(* CODESYS project sensata_pressuretransducers.library
   Company: Sensata Technologies
   Version: 0.0.1
   DocFormat: reStructuredText
   Placeholder: Sensata_PressureTransducers
   Title: Sensata_PressureTransducers

Project tree, tasks and I/O mapping:
  libraries: Sensata_Common, * (Sensata Technologies); Sensata_Utilities, * (Sensata Technologies); Tc2_Standard, * (Beckhoff Automation GmbH); Tc2_System, * (Beckhoff Automation GmbH); Tc2_Utilities, * (Beckhoff Automation GmbH); Tc3_Module, * (Beckhoff Automation GmbH)
  Abstract/
    function block FB_PressureTransducer [ST]: M_GetAlicatFlowData, M_GetPressure
  Concrete/
    Agilent/
      AgilentVacuumGauge/
        function block FB_AgilentVacuumGauge [ST]: M_Connect, M_Disconnect, M_GetConnectStatus, P_bConnectBusy, P_bConnected, P_strDescription, P_strMake, P_strModel, P_strVersion, M_GetPressure, A_CommandRecovery, M_RouterHelper
      data type E_Agilent_Error
    Alicat/
      AlicatAbsolute/
        function block FB_AlicatAbsolute [ST]: M_GetAlicatAbsData, M_LockDisplay, M_UnlockDisplay, M_Connect, M_Disconnect, M_GetConnectStatus, P_bConnectBusy, P_bConnected, P_strDescription, P_strMake, P_strModel, P_strVersion, M_GetPressure, A_CommandRecovery, M_RouterHelper
      AlicatDifferential/
        function block FB_AlicatDifferential [ST]: M_GetAlicatDiffData, M_LockDisplay, M_Tare, M_UnlockDisplay, M_Connect, M_Disconnect, M_GetConnectStatus, P_bConnectBusy, P_bConnected, P_strDescription, P_strMake, P_strModel, P_strVersion, M_GetPressure, A_CommandRecovery, M_RouterHelper
      AlicatFlowMeter/
        function block FB_AlicatFlowMeter [ST]: M_GetAlicatFlowData, M_LockDisplay, M_Tare, M_UnlockDisplay, M_Connect, M_Disconnect, M_GetConnectStatus, P_bConnectBusy, P_bConnected, P_strDescription, P_strMake, P_strModel, P_strVersion, M_GetPressure, A_CommandRecovery, M_RouterHelper
      data type E_Alicat_Error
    Structures/
      data type ST_AlicatAbsoluteDataFrame
      data type ST_AlicatDifferentialDataFrame
      data type ST_AlicatFlowMeter
      data type ST_SerialDataFrame
  Interfaces/
    interface I_PressureSensing: M_GetPressure
  Project Information/
    function F_GetCompany [ST]
    function F_GetTitle [ST]
    function F_GetVersion [ST]
  Version/
    global variables Global_Version
*)

// Concrete/Agilent/E_Agilent_Error
{attribute 'qualified_only'}
{attribute 'strict'}
TYPE E_Agilent_Error :
(
	None := 0,
	
	CommandRouterError			:= 0100,  // Error on the command router FB
	CommandFault 				:= 0101, // Command failed to execute
	
	FailedToConnect 			:= 0200, // Connect command failed
	FailedToDisconnect 			:= 0201, // Disonnect command failed
	FailedToGetConnectStatus 	:= 0202, // GetConnectStatus command failed
	
	FailedToReadSerialData		:= 0203,   // ReadSerialDataFrame from Agilent failed
	
	FailedToLoadProgram			:= 0300, // LoadProgram command failed
	FailedToGetCurrentProgram	:= 0301, // GetCurrentProgram command failed
	FailedToStartProgram		:= 0302, // StartProgram command failed
	FailedToStopProgram			:= 0303, // StopProgram command failed
	FailedToPauseProgram		:= 0304, // PauseProgram command failed
	FailedToGetProgramState		:= 0305, // GetProgramState command failed
	
	FailedToEnable				:= 0400, // Enable command failed
	FailedToDisable				:= 0401, // Disable command failed
	FailedToGetEnableStatus		:= 0402, // GetEnableStatus command failed
	
	FailedToPowerOn				:= 0500, // PowerOn command failed
	FailedToPowerOff			:= 0501, // PowerOff command failed
	FailedToGetPowerStatus		:= 0502, // GetPowerStatus command failed
	
	FailedToReset				:= 0600, // Reset command failed

	FailedToGetSafetyStatus		:= 0700 // GetSafetyStatus command failed
) UDINT;
END_TYPE

// Concrete/Alicat/E_Alicat_Error
{attribute 'qualified_only'}
{attribute 'strict'}
TYPE E_Alicat_Error :
(
	None := 0,
	
	CommandRouterError			:= 0100,  // Error on the command router FB
	CommandFault 				:= 0101, // Command failed to execute
	
	FailedToConnect 			:= 0200, // Connect command failed
	FailedToDisconnect 			:= 0201, // Disonnect command failed
	FailedToGetConnectStatus 	:= 0202, // GetConnectStatus command failed
	
	FailedToReadSerialData		:= 0203,   // ReadSerialDataFrame from Alicat failed
	FailedToLockDisplay			:= 0204,   // LockDisplay of AlicatDevice failed
	FailedToUnlockDisplay		:= 0205,   // UnlockDisplay of AlicatDevice failed
	FailedToTareDifferentialGauge := 0206, //Taring Differential Pressure Transducer failed
	FailedToTareFlowMeter 		:= 0207,   //Taring Flow Meter failed
	
	FailedToLoadProgram			:= 0300, // LoadProgram command failed
	FailedToGetCurrentProgram	:= 0301, // GetCurrentProgram command failed
	FailedToStartProgram		:= 0302, // StartProgram command failed
	FailedToStopProgram			:= 0303, // StopProgram command failed
	FailedToPauseProgram		:= 0304, // PauseProgram command failed
	FailedToGetProgramState		:= 0305, // GetProgramState command failed
	
	FailedToEnable				:= 0400, // Enable command failed
	FailedToDisable				:= 0401, // Disable command failed
	FailedToGetEnableStatus		:= 0402, // GetEnableStatus command failed
	
	FailedToPowerOn				:= 0500, // PowerOn command failed
	FailedToPowerOff			:= 0501, // PowerOff command failed
	FailedToGetPowerStatus		:= 0502, // GetPowerStatus command failed
	
	FailedToReset				:= 0600, // Reset command failed

	FailedToGetSafetyStatus		:= 0700 // GetSafetyStatus command failed
) UDINT;
END_TYPE

// Concrete/Structures/ST_AlicatAbsoluteDataFrame
TYPE ST_AlicatAbsoluteDataFrame :
STRUCT
	strDeviceID : STRING;
	lrAbsPressure : LREAL;
	strStatusCode : STRING;	
END_STRUCT
END_TYPE

// Concrete/Structures/ST_AlicatDifferentialDataFrame
TYPE ST_AlicatDifferentialDataFrame :
STRUCT
	strDeviceID : STRING;
	lrDiffPressure : LREAL;
	strStatusCode : STRING;	
END_STRUCT
END_TYPE

// Concrete/Structures/ST_AlicatFlowMeter
TYPE ST_AlicatFlowMeter :
STRUCT
	strDeviceID     : STRING;
	lrAbsPressure   : LREAL;
	lrTemperature   : LREAL;
	lrVolFlowRate   : LREAL;
	lrMassFlowRate  : LREAL;
	lrTotalizedFlow : LREAL;
	strGasSelect    : STRING;
	strStatusCode   : STRING;
END_STRUCT
END_TYPE

// Concrete/Structures/ST_SerialDataFrame
TYPE ST_SerialDataFrame :
STRUCT
	stAlicatAbs : ST_AlicatAbsoluteDataFrame;
	stAlicatDiff : ST_AlicatDifferentialDataFrame;
	stAlicatFlow : ST_AlicatFlowMeter;
END_STRUCT
END_TYPE

// Version/Global_Version
{attribute 'TcGenerated'}
{attribute 'no-analysis'}
{attribute 'linkalways'}
// This function has been automatically generated from the project information.
VAR_GLOBAL CONSTANT
	{attribute 'const_non_replaced'}
	stLibVersion_Sensata_PressureTransducers : ST_LibVersion := (iMajor := 0, iMinor := 0, iBuild := 1, iRevision := 0, nFlags := 0, sVersion := '0.0.1');
END_VAR

// Abstract/FB_PressureTransducer
FUNCTION_BLOCK FB_PressureTransducer EXTENDS FB_Device IMPLEMENTS I_PressureSensing
VAR_INPUT
END_VAR
VAR_OUTPUT
END_VAR
VAR
END_VAR

METHOD M_GetAlicatFlowData : BOOL

VAR_OUTPUT
		(*_output/input_datatypeName*)
	_out_lrealPressure	   : LREAL;
	_out_lrealTotFlow      : LREAL;
	_out_lrealMassFlowRate : LREAL;
	_out_lrealVolFlowRate  : LREAL;
	_out_stResult : ST_SerialDataFrame;
END_VAR
M_GetAlicatFlowData := TRUE;
THIS^.M_LogWarning('M_GetAlicatFlowData not implemented');
END_METHOD

METHOD M_GetPressure : BOOL
VAR_OUTPUT
	(*_output/input_datatypeName*)
	_out_lrealPressure	: LREAL;
END_VAR
M_GetPressure := TRUE;
THIS^.M_LogWarning('M_GetPressure not implemented');
END_METHOD

END_FUNCTION_BLOCK

// Interfaces/I_PressureSensing
INTERFACE I_PressureSensing

METHOD M_GetPressure : BOOL
VAR_INPUT
END_VAR
VAR_OUTPUT
	_out_lrealPressure : LREAL; //_output/input_datatypeName
END_VAR
END_METHOD

END_INTERFACE

// Concrete/Agilent/AgilentVacuumGauge/FB_AgilentVacuumGauge
FUNCTION_BLOCK FB_AgilentVacuumGauge EXTENDS FB_PressureTransducer IMPLEMENTS I_PressureSensing, I_Connectable, I_DeviceInfo
VAR_INPUT
	in_fbApi : REFERENCE TO FB_CommandRouter;
END_VAR
VAR_OUTPUT
END_VAR
VAR
	//Copied all the variables from UReSeries program - still not sure which all we need
	bConnected: BOOL; // Value of P_bConnected
	bEnabled: BOOL; // Value of P_bEnabled
	bPoweredOn: BOOL; // Value of P_bPoweredOn
	strLoadedProgram: STRING(255); // Value of P_strLoadedProgram
	enumProgramState: E_PROGRAMSTATE; // Value of P_enumProgramState
	bRouterBusy: BOOL; // TRUE while M_RouterHelper is being used by a method
	bResetBusy: BOOL; // Value of P_bResetBusy
	
	//ST Adding parameters below
	bDisconnected: BOOL;
	bGetPressureSuccessful: BOOL;
	
	//Command Steps
	intGetPressureStep		 : INT;
	intConnectStep	  		 : INT;
	intDisconnectStep 		 : INT;
	intRouterHelperStep		: INT;
		
	//CommandBusy Bits
	bGetPressureBusy 	   : BOOL;
	bConnectBusy	 	   : BOOL;
	bDisconnectBusy  	   : BOOL;
	bRouterHelperBusy	   : BOOL;
END_VAR

A_CommandRecovery();

(* This method should establish any external connections required to use the
	functions of the device, and return TRUE and set P_bConnected to TRUE once
	connected. *)
METHOD M_Connect : BOOL
VAR CONSTANT
	_strCOMMAND_NAME : T_MaxString	:= 'Connect'; // Name of the API method
	_timeCOMMAND_TIMEOUT : TIME		:= T#100S; // Max time to receive API response
	_strSTART_MSG : T_MaxString		:= 'Connecting'; // Prints when method starts
	_strEND_MSG : T_MaxString		:= 'Connected'; // Prints when method finishes
	_udintERROR_ID : UDINT			:= E_Agilent_Error.FailedToConnect; // Error ID to set if command fails
	_strERROR_MSG : T_MaxString		:= 'Failed to connect to Agilent Vacuum Gauge!'; // Error message to set if command fails
END_VAR
VAR_INST
	_inst_arrParams: T_ApiParameterList; // Parameters array
	_inst_arrOutputs: T_ApiParameterList; // Outputs array
	_inst_strRet: T_ApiParamValue; // Return string from the router
	_inst_intStep: INT; // Current method step
	_inst_fbParams: FB_ApiParamBuilder; // Parameter builder FB
END_VAR
VAR
	_bComplete: BOOL; // True if the routing finishes
	_intRet: INT; // Return string converted to an integer
	_bResult : BOOL; // Output of the method
END_VAR
_inst_intStep := intConnectStep;
bConnectBusy  := TRUE;

_bResult := FALSE;
CASE _inst_intStep OF
	0: // Wait for no error and router not busy
		IF NOT THIS^.P_bError AND NOT bRouterBusy THEN
			bRouterBusy := TRUE;
			_inst_intStep := _inst_intStep + 10;
		END_IF
		
	10: // Initialize parameters
		THIS^.M_LogMessage(_strSTART_MSG);
		_inst_fbParams.M_ClearParameters();
		// ADD ANY PARAMETERS HERE
		_inst_fbParams.M_OutputToParameterList(_inst_arrParams);
		_inst_intStep := _inst_intStep + 10;
		
	20: // Route the command
		_bComplete := M_RouterHelper(
			_in_strMethodName := _strCOMMAND_NAME, 
			_in_timeTimeout := _timeCOMMAND_TIMEOUT,
			_inout_arrParams := _inst_arrParams,
			_inout_arrOutputs := _inst_arrOutputs,
			_out_strReturnValue=>_inst_strRet);
		
		// If route completed, move to next step
		IF _bComplete THEN
			_inst_intStep := _inst_intStep + 10;
			bRouterBusy := FALSE;
		ELSIF THIS^.P_bError THEN
			_inst_intStep := 0;
			bRouterBusy := FALSE;
		END_IF
		
	30: // Parse results
		_intRet := STRING_TO_INT(_inst_strRet);
		IF _intRet > 0 THEN
			_bResult := TRUE;
			THIS^.M_LogMessage(_strEND_MSG);
			// DO ANY PARSING HERE
			bConnected := TRUE;
			
		// Set error if command failed
		ELSE
			THIS^.M_SetError(_udintERROR_ID, _strERROR_MSG);
		END_IF
		
		// Go back to start
		_inst_intStep := 0;
END_CASE
M_Connect := _bResult;
intConnectStep := _inst_intStep;
END_METHOD

(* This method should break any connections established by M_Connect. It should
	immediately set P_bConnected to false unless all connections are known to
	be still active, and return TRUE once those connections are all fully
	disconnected. *)
METHOD M_Disconnect : BOOL
VAR CONSTANT
	_strCOMMAND_NAME : T_MaxString	:= 'Disconnect'; // Name of the API method
	_timeCOMMAND_TIMEOUT : TIME		:= T#30S; // Max time to receive API response
	_strSTART_MSG : T_MaxString		:= 'Disconnecting'; // Prints when method starts
	_strEND_MSG : T_MaxString		:= 'Disconnected'; // Prints when method finishes
	_udintERROR_ID : UDINT			:= E_Agilent_Error.FailedToDisconnect; // Error ID to set if command fails
	_strERROR_MSG : T_MaxString		:= 'Failed to disconnect from AgilentVacuumGauge!'; // Error message to set if command fails
END_VAR
VAR_INST
	_inst_arrParams: T_ApiParameterList; // Parameters array
	_inst_arrOutputs: T_ApiParameterList; // Outputs array
	_inst_strRet: T_ApiParamValue; // Return string from the router
	_inst_intStep: INT; // Current method step
	_inst_fbParams: FB_ApiParamBuilder; // Parameter builder FB
END_VAR
VAR
	_bComplete: BOOL; // True if the routing finishes
	_intRet: INT; // Return string converted to an integer
	_bResult : BOOL; // Output of the method
END_VAR
_inst_intStep := intDisconnectStep;
bDisconnectBusy := TRUE;

_bResult := FALSE;
CASE _inst_intStep OF
	0: // Wait for no error and router not busy
		IF NOT THIS^.P_bError AND NOT bRouterBusy THEN
			bRouterBusy := TRUE;
			_inst_intStep := _inst_intStep + 10;
		END_IF
		
	10: // Initialize parameters
		THIS^.M_LogMessage(_strSTART_MSG);
		_inst_fbParams.M_ClearParameters();
		// ADD ANY PARAMETERS HERE
		_inst_fbParams.M_OutputToParameterList(_inst_arrParams);
		_inst_intStep := _inst_intStep + 10;
		
	20: // Route the command
		_bComplete := M_RouterHelper(
			_in_strMethodName := _strCOMMAND_NAME, 
			_in_timeTimeout := _timeCOMMAND_TIMEOUT,
			_inout_arrParams := _inst_arrParams,
			_inout_arrOutputs := _inst_arrOutputs,
			_out_strReturnValue=>_inst_strRet);
		
		// If route completed, move to next step
		IF _bComplete THEN
			_inst_intStep := _inst_intStep + 10;
			bRouterBusy := FALSE;
		ELSIF THIS^.P_bError THEN
			_inst_intStep := 0;
			bRouterBusy := FALSE;
		END_IF
		
	30: // Parse results
		_intRet := STRING_TO_INT(_inst_strRet);
		IF _intRet > 0 THEN
			_bResult := TRUE;
			THIS^.M_LogMessage(_strEND_MSG);
			// DO ANY PARSING HERE
			bConnected := FALSE;
			
		// Set error if command failed
		ELSE
			THIS^.M_SetError(_udintERROR_ID, _strERROR_MSG);
		END_IF
		
		// Go back to start
		_inst_intStep := 0;
END_CASE
M_Disconnect := _bResult;
intDisconnectStep := _inst_intStep;
END_METHOD

(* This method should explicitly check the connection status of the device.
	Once the connection status is known, this method should return TRUE.
	If this method fails, P_bConnected should be set to FALSE since the device
	is not absolutely known to still be connected. *)
METHOD M_GetConnectStatus : BOOL
VAR_OUTPUT
	(* This should return TRUE if all connections required to make the device
		function properly are known to be connected, and FALSE otherwise. *)
	bConnected	: BOOL;
END_VAR
bConnected := P_bConnected;
M_GetConnectStatus := TRUE;
THIS^.M_LogWarning('Get connect status not implemented in FB_AgilentVacuumGauge!');
END_METHOD

(* This property should be TRUE while any method in this interface is actively
	executing, or FALSE otherwise. *)
PROPERTY P_bConnectBusy : BOOL
GET
END_GET
END_PROPERTY

(* This should be set to TRUE if M_Connect is successful or M_GetConnectStatus
	determines the device to be connected, and set to FALSE if M_Disconnect is
	called at all, M_GetConnectStatus fails, or M_GetConnectStatus determines
	the device to be not connected. *)
PROPERTY P_bConnected : BOOL
GET
END_GET
END_PROPERTY

PROPERTY P_strDescription : Sensata_Common.T_MaxString
GET
END_GET
END_PROPERTY

PROPERTY P_strMake : Sensata_Common.T_MaxString
GET
END_GET
END_PROPERTY

PROPERTY P_strModel : Sensata_Common.T_MaxString
GET
END_GET
END_PROPERTY

PROPERTY P_strVersion : Sensata_Common.T_MaxString
GET
END_GET
END_PROPERTY

METHOD M_GetPressure : BOOL
VAR_OUTPUT
	(*_output/input_datatypeName*)
	_out_lrealPressure	: LREAL;
END_VAR
VAR CONSTANT
	_strCOMMAND_NAME : T_MaxString	:= 'GetPressure'; // Name of the API method
	_timeCOMMAND_TIMEOUT : TIME		:= T#5S; // Max time to receive API response
	_strSTART_MSG : T_MaxString		:= 'Reading Pressure Value'; // Prints when method starts
	_strEND_MSG : T_MaxString		:= 'Pressure Read'; // Prints when method finishes
	_udintERROR_ID : UDINT			:= E_Agilent_Error.FailedToReadSerialData; // Error ID to set if command fails
	_strERROR_MSG : T_MaxString		:= 'Failed to read serial data and hence pressure!'; // Error message to set if command fails
END_VAR
VAR_INST
	_inst_arrParams: T_ApiParameterList; // Parameters array
	_inst_arrOutputs: T_ApiParameterList; // Outputs array
	_inst_strRet: T_ApiParamValue; // Return string from the router
	_inst_intStep: INT; // Current method step
	_inst_fbParams: FB_ApiParamBuilder; // Parameter builder FB
END_VAR
VAR
	_bComplete: BOOL; // True if the routing finishes
	_intRet: INT; // Return string converted to an integer
	_bResult : BOOL; // Output of the method
END_VAR
_inst_intStep := intGetPressureStep;
bGetPressureBusy := TRUE;

_bResult := FALSE;
CASE _inst_intStep OF
	0: // Wait for no error and router not busy
		IF NOT THIS^.P_bError AND NOT bRouterBusy THEN
			bRouterBusy := TRUE;
			_inst_intStep := _inst_intStep + 10;
		END_IF
		
	10: // Initialize parameters
		THIS^.M_LogMessage(_strSTART_MSG);
		_inst_fbParams.M_ClearParameters();
		// ADD ANY PARAMETERS HERE
		_inst_fbParams.M_OutputToParameterList(_inst_arrParams);
		_inst_intStep := _inst_intStep + 10;
		
	20: // Route the command
		_bComplete := M_RouterHelper(
			_in_strMethodName := _strCOMMAND_NAME, 
			_in_timeTimeout := _timeCOMMAND_TIMEOUT,
			_inout_arrParams := _inst_arrParams,
			_inout_arrOutputs := _inst_arrOutputs,
			_out_strReturnValue=>_inst_strRet);
		
		// If route completed, move to next step
		IF _bComplete THEN
			_inst_intStep := _inst_intStep + 10;
			bRouterBusy := FALSE;
		ELSIF THIS^.P_bError THEN
			_inst_intStep := 0;
			bRouterBusy := FALSE;
		END_IF
		
	30: // Parse results
		_intRet := STRING_TO_INT(_inst_strRet);
		IF _intRet > 0 THEN
			_bResult := TRUE;
			THIS^.M_LogMessage(_strEND_MSG);
			// DO ANY PARSING HERE
			_out_lrealPressure := _inst_fbParams.M_ParseDouble(_inst_fbParams.M_GetParameter('Pressure'));
//			_inst_fbParams.M_LoadFromParameterList(_inst_arrOutputs);
//			bEnabled := _inst_fbParams.M_ParseBool(_inst_fbParams.M_GetParameter('enabled'));
//			THIS^.bEnabled := bEnabled;			
			
		// Set error if command failed
		ELSE
			THIS^.M_SetError(_udintERROR_ID, _strERROR_MSG);
		END_IF
		
		// Go back to start
		_inst_intStep := 0;
END_CASE
M_GetPressure := _bResult;
intGetPressureStep := _inst_intStep;
END_METHOD

ACTION A_CommandRecovery:
IF NOT bGetPressureBusy AND intGetPressureStep > 0 THEN
	intGetPressureStep := 0;
	bRouterBusy := FALSE;
	THIS^.M_LogWarning('Get Pressure ended prematurely!');
END_IF
bGetPressureBusy := FALSE;

IF NOT bConnectBusy AND intConnectStep > 0 THEN
	intConnectStep := 0;
	bRouterBusy := FALSE;
	THIS^.M_LogWarning('Connect ended prematurely!');
END_IF
bConnectBusy := FALSE;

IF NOT bDisconnectBusy AND intDisconnectStep > 0 THEN
	intDisconnectStep := 0;
	bRouterBusy := FALSE;
	THIS^.M_LogWarning('Disconnect ended prematurely!');
END_IF
bDisconnectBusy := FALSE;

IF NOT bRouterHelperBusy AND intRouterHelperStep > 0 THEN
	intRouterHelperStep := 0;
	THIS^.M_LogWarning('Router helper ended prematurely!');
END_IF
bRouterHelperBusy := FALSE;
END_ACTION

(*
Sends the given method to the API and receives and partially parses the result.
*)
METHOD PRIVATE M_RouterHelper : BOOL
VAR_INPUT
	(* Name of the method to call. *)
	_in_strMethodName : T_MaxString;
	(* Maximum time to wait for method response. *)
	_in_timeTimeout : TIME;
END_VAR
VAR_IN_OUT
	(* The array of parameters to send to the API. *)
	_inout_arrParams : T_ApiParameterList;
	(* The array that gets populated with any method output data. *)
	_inout_arrOutputs : T_ApiParameterList;
END_VAR
VAR_OUTPUT
	(* JSON string of the method return value. *)
	_out_strReturnValue: T_ApiParamValue;
END_VAR
VAR_INST
	(* Current step. *)
	_inst_intStep: INT;
	(* True if the method executed. *)
	_inst_bExec: BOOL;
	(* Return string of the method. *)
	_inst_strRet: T_ApiParamValue;
END_VAR
VAR
	(* True once the command routing finishes. *)
	_bComplete: BOOL;
	(* True once the API connects. *)
	_bApiConnect: BOOL;
END_VAR
_inst_intStep := intRouterHelperStep;
bRouterHelperBusy := TRUE;

CASE _inst_intStep OF
	0: // Start process only if there is no error on this FB
		IF NOT THIS^.P_bError THEN
			_inst_intStep := 10;
		END_IF
		
	10: // Check if command router connected
		IF NOT in_fbApi.P_bConnected THEN
			_inst_intStep := 20; // Go to API connect step
		ELSE
			_inst_intStep := 30; // Go to route command step
		END_IF
		
	20: // Connect the command router
		_bApiConnect := in_fbApi.M_Connect();
		IF _bApiConnect THEN
			_inst_intStep := _inst_intStep + 10; // Go to next step
		ELSIF in_fbApi.P_bError THEN
			THIS^.M_SetError(E_Agilent_Error.CommandRouterError, 'Error on command router function block while connecting!');
			_inst_intStep := 0; // Go back to start
		END_IF
		
	30:	// Route the command
		_bComplete := in_fbApi.M_RouteCommand(
			_in_strModuleId := in_strUniqueId,
			_in_strMethodName := _in_strMethodName,
			_in_timeTimeout := _in_timeTimeout,
			_inout_arrParameters := _inout_arrParams,
			_inout_arrOutputs := _inout_arrOutputs,
			_out_bCommandExecuted => _inst_bExec,
			_out_strReturnValue => _inst_strRet);
		IF _bComplete THEN
			_inst_intStep := _inst_intStep + 10; // Go to next step
		ELSIF in_fbApi.P_bError THEN
			THIS^.M_SetError(E_Agilent_Error.CommandRouterError, 'Error on command router function block while routing command!');
			_inst_intStep := 0; // Go back to start
		END_IF
		
	40: // Check result then go back to start
		IF NOT _inst_bExec THEN
			THIS^.M_SetError(E_Agilent_Error.CommandFault, 'Method in API failed to execute!');
		ELSE
			_out_strReturnValue := _inst_strRet;
			M_RouterHelper := TRUE;
		END_IF
		_inst_intStep := 0; // Go back to start
END_CASE
intRouterHelperStep := _inst_intStep;
END_METHOD

END_FUNCTION_BLOCK

// Concrete/Alicat/AlicatAbsolute/FB_AlicatAbsolute
FUNCTION_BLOCK FB_AlicatAbsolute EXTENDS FB_PressureTransducer IMPLEMENTS I_PressureSensing, I_Connectable, I_DeviceInfo
VAR_INPUT
	in_fbApi : REFERENCE TO FB_CommandRouter;
END_VAR
VAR_OUTPUT
END_VAR
VAR
	//Copied all the variables from UReSeries program - still not sure which all we need
	bConnected: BOOL; // Value of P_bConnected
	bEnabled: BOOL; // Value of P_bEnabled
	bPoweredOn: BOOL; // Value of P_bPoweredOn
	strLoadedProgram: STRING(255); // Value of P_strLoadedProgram
	enumProgramState: E_PROGRAMSTATE; // Value of P_enumProgramState
	bRouterBusy: BOOL; // TRUE while M_RouterHelper is being used by a method
	bResetBusy: BOOL; // Value of P_bResetBusy
	//ST Adding parameters below
	bDisconnected: BOOL;
	bGetPressureSuccessful: BOOL;
	bGetAlicatDataSuccessful: BOOL;
	bLockDisplaySuccessful: BOOL;
	bUnlockDisplaySuccessful: BOOL;
	
	//Command Steps
	intGetPressureStep		 : INT;
	intConnectStep	  		 : INT;
	intDisconnectStep 		 : INT;
	intGetAlicatAbsDataStep : INT;
	intLockDisplayStep		 : INT;
	intUnlockDisplayStep	 : INT;
	intTareStep			  	 : INT;
	intRouterHelperStep	     : INT;
	
	
	//CommandBusy Bits
	bGetPressureBusy 	   : BOOL;
	bConnectBusy	 	   : BOOL;
	bDisconnectBusy  	   : BOOL;
	bGetAlicatAbsDataBusy  : BOOL;
	bLockDisplayBusy	   : BOOL;
	bUnlockDisplayBusy	   : BOOL;
	bTareBusy			   : BOOL;
	bRouterHelperBusy	   : BOOL;
	
END_VAR

A_CommandRecovery();

(* This method returns the Pressure Value from the Alicat Absolute Pressure Gauge.
Once the Pressure value is obtained, this method must return TRUE*)
METHOD M_GetAlicatAbsData : BOOL
VAR_OUTPUT
	(*_output/input_datatypeName*)
	_out_lrealPressure	: LREAL;
	_out_stResult : ST_SerialDataFrame;
END_VAR
VAR CONSTANT
	_strCOMMAND_NAME : T_MaxString	:= 'GetAlicatAbsData'; // Name of the API method
	_timeCOMMAND_TIMEOUT : TIME		:= T#5S; // Max time to receive API response
	_strSTART_MSG : T_MaxString		:= 'Reading Alicat Serial Frame'; // Prints when method starts
	_strEND_MSG : T_MaxString		:= 'Read Alicat Serial Frame successfully'; // Prints when method finishes
	_udintERROR_ID : UDINT			:= E_Alicat_Error.FailedToReadSerialData; // Error ID to set if command fails
	_strERROR_MSG : T_MaxString		:= 'Failed to read Alicat Serial Frame!'; // Error message to set if command fails
END_VAR
VAR_INST
	_inst_arrParams: T_ApiParameterList; // Parameters array
	_inst_arrOutputs: T_ApiParameterList; // Outputs array
	_inst_strRet: T_ApiParamValue; // Return string from the router
	_inst_intStep: INT; // Current method step
	_inst_fbParams: FB_ApiParamBuilder; // Parameter builder FB
END_VAR
VAR
	_bComplete: BOOL; // True if the routing finishes
	_intRet: INT; // Return string converted to an integer
	_bResult : BOOL; // Output of the method
	_pStructPointer : PVOID; // Pointer to the struct
	_pStructPointerAbs : PVOID; 
END_VAR
VAR_INPUT
	
END_VAR
_inst_intStep := intGetAlicatAbsDataStep;
bGetAlicatAbsDataBusy := TRUE;

_bResult := FALSE;
CASE _inst_intStep OF
	0: // Wait for no error and router not busy
		IF NOT THIS^.P_bError AND NOT bRouterBusy THEN
			bRouterBusy := TRUE;
			_inst_intStep := _inst_intStep + 10;
		END_IF
		
	10: // Initialize parameters
		THIS^.M_LogMessage(_strSTART_MSG);
		_inst_fbParams.M_ClearParameters();
		// ADD ANY PARAMETERS HERE
		_inst_fbParams.M_OutputToParameterList(_inst_arrParams);
		_inst_intStep := _inst_intStep + 10;
		
	20: // Route the command
		_bComplete := M_RouterHelper(
			_in_strMethodName := _strCOMMAND_NAME, 
			_in_timeTimeout := _timeCOMMAND_TIMEOUT,
			_inout_arrParams := _inst_arrParams,
			_inout_arrOutputs := _inst_arrOutputs,
			_out_strReturnValue=>_inst_strRet);
		
		// If route completed, move to next step
		IF _bComplete THEN
			_inst_intStep := _inst_intStep + 10;
			bRouterBusy := FALSE;
		ELSIF THIS^.P_bError THEN
			_inst_intStep := 0;
			bRouterBusy := FALSE;
		END_IF
		
	30: // Parse results
		_intRet := STRING_TO_INT(_inst_strRet);
		IF _intRet > 0 THEN
			_bResult := TRUE;
			THIS^.M_LogMessage(_strEND_MSG);
			// DO ANY PARSING HERE
			_pStructPointer := _inst_fbParams.M_GetParameter('alicatAbsDataFrame');	//Because this is the name of the parameter on the API side - type doesn't matter?
			
			_pStructPointerAbs := _inst_fbParams.M_GetStructMember(_pStructPointer, 'AlicatAbsoluteDataFrame');	//Because AlicatAbsoluteDataFrame is a member of the main struct on the API side			
		
			_out_stResult.stAlicatAbs.strDeviceID := _inst_fbParams.M_ParseString(_inst_fbParams.M_GetStructMember(_pStructPointerAbs, 'DeviceID'));
			_out_stResult.stAlicatAbs.lrAbsPressure := _inst_fbParams.M_ParseDouble(_inst_fbParams.M_GetStructMember(_pStructPointerAbs, 'AbsPressure'));
			_out_stResult.stAlicatAbs.strStatusCode := _inst_fbParams.M_ParseString(_inst_fbParams.M_GetStructMember(_pStructPointerAbs, 'StatusCode'));
			
			_out_lrealPressure := _out_stResult.stAlicatAbs.lrAbsPressure;
			
//			_inst_fbParams.M_LoadFromParameterList(_inst_arrOutputs);
//			bConnected := _inst_fbParams.M_ParseBool(_inst_fbParams.M_GetParameter('connected'));
//			THIS^.bConnected := bConnected;
			
		// Set error if command failed
		ELSE
			THIS^.M_SetError(_udintERROR_ID, _strERROR_MSG);
		END_IF
		
		// Go back to start
		_inst_intStep := 0;
END_CASE
M_GetAlicatAbsData := _bResult;
intGetAlicatAbsDataStep := _inst_intStep;
END_METHOD

(* This method returns the status of whether the screen on the device has been locked.
Once the screen is locked, this method must return TRUE*)
METHOD M_LockDisplay : BOOL
VAR_INPUT
END_VAR
VAR CONSTANT
	_strCOMMAND_NAME : T_MaxString	:= 'LockDisplay'; // Name of the API method
	_timeCOMMAND_TIMEOUT : TIME		:= T#2S; // Max time to receive API response
	_strSTART_MSG : T_MaxString		:= 'Locking Alicat Display'; // Prints when method starts
	_strEND_MSG : T_MaxString		:= 'Locked Alicat Display'; // Prints when method finishes
	_udintERROR_ID : UDINT			:= E_Alicat_Error.FailedToLockDisplay; // Error ID to set if command fails
	_strERROR_MSG : T_MaxString		:= 'Failed to lock display!'; // Error message to set if command fails
END_VAR
VAR_INST
	_inst_arrParams: T_ApiParameterList; // Parameters array
	_inst_arrOutputs: T_ApiParameterList; // Outputs array
	_inst_strRet: T_ApiParamValue; // Return string from the router
	_inst_intStep: INT; // Current method step
	_inst_fbParams: FB_ApiParamBuilder; // Parameter builder FB
END_VAR
VAR
	_bComplete: BOOL; // True if the routing finishes
	_intRet: INT; // Return string converted to an integer
	_bResult : BOOL; // Output of the method
END_VAR
_inst_intStep 	 := intLockDisplayStep;
bLockDisplayBusy := TRUE;

_bResult := FALSE;
CASE _inst_intStep OF
	0: // Wait for no error and router not busy
		IF NOT THIS^.P_bError AND NOT bRouterBusy THEN
			bRouterBusy := TRUE;
			_inst_intStep := _inst_intStep + 10;
		END_IF
		
	10: // Initialize parameters
		THIS^.M_LogMessage(_strSTART_MSG);
		_inst_fbParams.M_ClearParameters();
		// ADD ANY PARAMETERS HERE
		_inst_fbParams.M_OutputToParameterList(_inst_arrParams);
		_inst_intStep := _inst_intStep + 10;
		
	20: // Route the command
		_bComplete := M_RouterHelper(
			_in_strMethodName := _strCOMMAND_NAME, 
			_in_timeTimeout := _timeCOMMAND_TIMEOUT,
			_inout_arrParams := _inst_arrParams,
			_inout_arrOutputs := _inst_arrOutputs,
			_out_strReturnValue=>_inst_strRet);
		
		// If route completed, move to next step
		IF _bComplete THEN
			_inst_intStep := _inst_intStep + 10;
			bRouterBusy := FALSE;
		ELSIF THIS^.P_bError THEN
			_inst_intStep := 0;
			bRouterBusy := FALSE;
		END_IF
		
	30: // Parse results
		_intRet := STRING_TO_INT(_inst_strRet);
		IF _intRet > 0 THEN
			_bResult := TRUE;
			THIS^.M_LogMessage(_strEND_MSG);
			// DO ANY PARSING HERE
//			_inst_fbParams.M_LoadFromParameterList(_inst_arrOutputs);
//			bConnected := _inst_fbParams.M_ParseBool(_inst_fbParams.M_GetParameter('connected'));
//			THIS^.bConnected := bConnected;
			
		// Set error if command failed
		ELSE
			THIS^.M_SetError(_udintERROR_ID, _strERROR_MSG);
		END_IF
		
		// Go back to start
		_inst_intStep := 0;
END_CASE
M_LockDisplay := _bResult;
intLockDisplayStep := _inst_intStep;
END_METHOD

(* This method returns the status of whether the screen on the device has been locked.
Once the screen is locked, this method must return TRUE*)
METHOD M_UnlockDisplay : BOOL
VAR_INPUT
END_VAR
VAR CONSTANT
	_strCOMMAND_NAME : T_MaxString	:= 'UnlockDisplay'; // Name of the API method
	_timeCOMMAND_TIMEOUT : TIME		:= T#2S; // Max time to receive API response
	_strSTART_MSG : T_MaxString		:= 'Unlocking Alicat Display'; // Prints when method starts
	_strEND_MSG : T_MaxString		:= 'Unlocked Alicat Display'; // Prints when method finishes
	_udintERROR_ID : UDINT			:= E_Alicat_Error.FailedToUnlockDisplay; // Error ID to set if command fails
	_strERROR_MSG : T_MaxString		:= 'Failed to unlock display!'; // Error message to set if command fails
END_VAR
VAR_INST
	_inst_arrParams: T_ApiParameterList; // Parameters array
	_inst_arrOutputs: T_ApiParameterList; // Outputs array
	_inst_strRet: T_ApiParamValue; // Return string from the router
	_inst_intStep: INT; // Current method step
	_inst_fbParams: FB_ApiParamBuilder; // Parameter builder FB
END_VAR
VAR
	_bComplete: BOOL; // True if the routing finishes
	_intRet: INT; // Return string converted to an integer
	_bResult : BOOL; // Output of the method
END_VAR
_inst_intStep := intUnlockDisplayStep;
bUnlockDisplayBusy := TRUE;

_bResult := FALSE;
CASE _inst_intStep OF
	0: // Wait for no error and router not busy
		IF NOT THIS^.P_bError AND NOT bRouterBusy THEN
			bRouterBusy := TRUE;
			_inst_intStep := _inst_intStep + 10;
		END_IF
		
	10: // Initialize parameters
		THIS^.M_LogMessage(_strSTART_MSG);
		_inst_fbParams.M_ClearParameters();
		// ADD ANY PARAMETERS HERE
		_inst_fbParams.M_OutputToParameterList(_inst_arrParams);
		_inst_intStep := _inst_intStep + 10;
		
	20: // Route the command
		_bComplete := M_RouterHelper(
			_in_strMethodName := _strCOMMAND_NAME, 
			_in_timeTimeout := _timeCOMMAND_TIMEOUT,
			_inout_arrParams := _inst_arrParams,
			_inout_arrOutputs := _inst_arrOutputs,
			_out_strReturnValue=>_inst_strRet);
		
		// If route completed, move to next step
		IF _bComplete THEN
			_inst_intStep := _inst_intStep + 10;
			bRouterBusy := FALSE;
		ELSIF THIS^.P_bError THEN
			_inst_intStep := 0;
			bRouterBusy := FALSE;
		END_IF
		
	30: // Parse results
		_intRet := STRING_TO_INT(_inst_strRet);
		IF _intRet > 0 THEN
			_bResult := TRUE;
			THIS^.M_LogMessage(_strEND_MSG);
			// DO ANY PARSING HERE
//			_inst_fbParams.M_LoadFromParameterList(_inst_arrOutputs);
//			bConnected := _inst_fbParams.M_ParseBool(_inst_fbParams.M_GetParameter('connected'));
//			THIS^.bConnected := bConnected;
			
		// Set error if command failed
		ELSE
			THIS^.M_SetError(_udintERROR_ID, _strERROR_MSG);
		END_IF
		
		// Go back to start
		_inst_intStep := 0;
END_CASE
M_UnlockDisplay := _bResult;
intUnlockDisplayStep := _inst_intStep;
END_METHOD

(* This method should establish any external connections required to use the
	functions of the device, and return TRUE and set P_bConnected to TRUE once
	connected. *)
METHOD M_Connect : BOOL
VAR CONSTANT
	_strCOMMAND_NAME : T_MaxString	:= 'Connect'; // Name of the API method
	_timeCOMMAND_TIMEOUT : TIME		:= T#100S; // Max time to receive API response
	_strSTART_MSG : T_MaxString		:= 'Connecting'; // Prints when method starts
	_strEND_MSG : T_MaxString		:= 'Connected'; // Prints when method finishes
	_udintERROR_ID : UDINT			:= E_Alicat_Error.FailedToConnect; // Error ID to set if command fails
	_strERROR_MSG : T_MaxString		:= 'Failed to connect to Absolute Pressure Transducer!'; // Error message to set if command fails
END_VAR
VAR_INST
	_inst_arrParams: T_ApiParameterList; // Parameters array
	_inst_arrOutputs: T_ApiParameterList; // Outputs array
	_inst_strRet: T_ApiParamValue; // Return string from the router
	_inst_intStep: INT; // Current method step
	_inst_fbParams: FB_ApiParamBuilder; // Parameter builder FB
END_VAR
VAR
	_bComplete: BOOL; // True if the routing finishes
	_intRet: INT; // Return string converted to an integer
	_bResult : BOOL; // Output of the method
END_VAR
_inst_intStep := intConnectStep;
bConnectBusy  := TRUE;

_bResult := FALSE;
CASE _inst_intStep OF
	0: // Wait for no error and router not busy
		IF NOT THIS^.P_bError AND NOT bRouterBusy THEN
			bRouterBusy := TRUE;
			_inst_intStep := _inst_intStep + 10;
		END_IF
		
	10: // Initialize parameters
		THIS^.M_LogMessage(_strSTART_MSG);
		_inst_fbParams.M_ClearParameters();
		// ADD ANY PARAMETERS HERE
		_inst_fbParams.M_OutputToParameterList(_inst_arrParams);
		_inst_intStep := _inst_intStep + 10;
		
	20: // Route the command
		_bComplete := M_RouterHelper(
			_in_strMethodName := _strCOMMAND_NAME, 
			_in_timeTimeout := _timeCOMMAND_TIMEOUT,
			_inout_arrParams := _inst_arrParams,
			_inout_arrOutputs := _inst_arrOutputs,
			_out_strReturnValue=>_inst_strRet);
		
		// If route completed, move to next step
		IF _bComplete THEN
			_inst_intStep := _inst_intStep + 10;
			bRouterBusy := FALSE;
		ELSIF THIS^.P_bError THEN
			_inst_intStep := 0;
			bRouterBusy := FALSE;
		END_IF
		
	30: // Parse results
		_intRet := STRING_TO_INT(_inst_strRet);
		IF _intRet > 0 THEN
			_bResult := TRUE;
			THIS^.M_LogMessage(_strEND_MSG);
			// DO ANY PARSING HERE
			bConnected := TRUE;
			
		// Set error if command failed
		ELSE
			THIS^.M_SetError(_udintERROR_ID, _strERROR_MSG);
		END_IF
		
		// Go back to start
		_inst_intStep := 0;
END_CASE
M_Connect := _bResult;
intConnectStep := _inst_intStep;
END_METHOD

(* This method should break any connections established by M_Connect. It should
	immediately set P_bConnected to false unless all connections are known to
	be still active, and return TRUE once those connections are all fully
	disconnected. *)
METHOD M_Disconnect : BOOL
VAR CONSTANT
	_strCOMMAND_NAME : T_MaxString	:= 'Disconnect'; // Name of the API method
	_timeCOMMAND_TIMEOUT : TIME		:= T#30S; // Max time to receive API response
	_strSTART_MSG : T_MaxString		:= 'Disconnecting'; // Prints when method starts
	_strEND_MSG : T_MaxString		:= 'Disconnected'; // Prints when method finishes
	_udintERROR_ID : UDINT			:= E_Alicat_Error.FailedToDisconnect; // Error ID to set if command fails
	_strERROR_MSG : T_MaxString		:= 'Failed to disconnect from Absolute Pressure Transducer!'; // Error message to set if command fails
END_VAR
VAR_INST
	_inst_arrParams: T_ApiParameterList; // Parameters array
	_inst_arrOutputs: T_ApiParameterList; // Outputs array
	_inst_strRet: T_ApiParamValue; // Return string from the router
	_inst_intStep: INT; // Current method step
	_inst_fbParams: FB_ApiParamBuilder; // Parameter builder FB
END_VAR
VAR
	_bComplete: BOOL; // True if the routing finishes
	_intRet: INT; // Return string converted to an integer
	_bResult : BOOL; // Output of the method
END_VAR
_inst_intStep := intDisconnectStep;
bDisconnectBusy := TRUE;

_bResult := FALSE;
CASE _inst_intStep OF
	0: // Wait for no error and router not busy
		IF NOT THIS^.P_bError AND NOT bRouterBusy THEN
			bRouterBusy := TRUE;
			_inst_intStep := _inst_intStep + 10;
		END_IF
		
	10: // Initialize parameters
		THIS^.M_LogMessage(_strSTART_MSG);
		_inst_fbParams.M_ClearParameters();
		// ADD ANY PARAMETERS HERE
		_inst_fbParams.M_OutputToParameterList(_inst_arrParams);
		_inst_intStep := _inst_intStep + 10;
		
	20: // Route the command
		_bComplete := M_RouterHelper(
			_in_strMethodName := _strCOMMAND_NAME, 
			_in_timeTimeout := _timeCOMMAND_TIMEOUT,
			_inout_arrParams := _inst_arrParams,
			_inout_arrOutputs := _inst_arrOutputs,
			_out_strReturnValue=>_inst_strRet);
		
		// If route completed, move to next step
		IF _bComplete THEN
			_inst_intStep := _inst_intStep + 10;
			bRouterBusy := FALSE;
		ELSIF THIS^.P_bError THEN
			_inst_intStep := 0;
			bRouterBusy := FALSE;
		END_IF
		
	30: // Parse results
		_intRet := STRING_TO_INT(_inst_strRet);
		IF _intRet > 0 THEN
			_bResult := TRUE;
			THIS^.M_LogMessage(_strEND_MSG);
			// DO ANY PARSING HERE
			bConnected := FALSE;
			
		// Set error if command failed
		ELSE
			THIS^.M_SetError(_udintERROR_ID, _strERROR_MSG);
		END_IF
		
		// Go back to start
		_inst_intStep := 0;
END_CASE
M_Disconnect := _bResult;
intDisconnectStep := _inst_intStep;
END_METHOD

(* This method should explicitly check the connection status of the device.
	Once the connection status is known, this method should return TRUE.
	If this method fails, P_bConnected should be set to FALSE since the device
	is not absolutely known to still be connected. *)
METHOD M_GetConnectStatus : BOOL
VAR_OUTPUT
	(* This should return TRUE if all connections required to make the device
		function properly are known to be connected, and FALSE otherwise. *)
	bConnected	: BOOL;
END_VAR
bConnected := P_bConnected;
M_GetConnectStatus := TRUE;
THIS^.M_LogWarning('Get connect status not implemented in FB_Absolute!');
END_METHOD

(* This property should be TRUE while any method in this interface is actively
	executing, or FALSE otherwise. *)
PROPERTY P_bConnectBusy : BOOL
GET
P_bConnectBusy := bRouterBusy;
END_GET
END_PROPERTY

(* This should be set to TRUE if M_Connect is successful or M_GetConnectStatus
	determines the device to be connected, and set to FALSE if M_Disconnect is
	called at all, M_GetConnectStatus fails, or M_GetConnectStatus determines
	the device to be not connected. *)
PROPERTY P_bConnected : BOOL
GET
P_bConnected := bConnected;
END_GET
END_PROPERTY

PROPERTY P_strDescription : Sensata_Common.T_MaxString
GET
END_GET
END_PROPERTY

PROPERTY P_strMake : Sensata_Common.T_MaxString
GET
END_GET
END_PROPERTY

PROPERTY P_strModel : Sensata_Common.T_MaxString
GET
END_GET
END_PROPERTY

PROPERTY P_strVersion : Sensata_Common.T_MaxString
GET
END_GET
END_PROPERTY

(* This method returns the Pressure Value from the Alicat Absolute Pressure Gauge.
Once the Pressure value is obtained, this method must return TRUE*)
METHOD M_GetPressure : BOOL
VAR_OUTPUT
	(*_output/input_datatypeName*)
	_out_lrealPressure	: LREAL;

END_VAR
VAR CONSTANT
	_strCOMMAND_NAME : T_MaxString	:= 'GetPressure'; // Name of the API method
	_timeCOMMAND_TIMEOUT : TIME		:= T#5S; // Max time to receive API response
	_strSTART_MSG : T_MaxString		:= 'Reading Pressure Value'; // Prints when method starts
	_strEND_MSG : T_MaxString		:= 'Pressure Read'; // Prints when method finishes
	_udintERROR_ID : UDINT			:= E_Alicat_Error.FailedToReadSerialData; // Error ID to set if command fails
	_strERROR_MSG : T_MaxString		:= 'Failed to read serial data and hence pressure!'; // Error message to set if command fails
END_VAR
VAR_INST
	_inst_arrParams: T_ApiParameterList; // Parameters array
	_inst_arrOutputs: T_ApiParameterList; // Outputs array
	_inst_strRet: T_ApiParamValue; // Return string from the router
	_inst_intStep: INT; // Current method step
	_inst_fbParams: FB_ApiParamBuilder; // Parameter builder FB
END_VAR
VAR
	_bComplete: BOOL; // True if the routing finishes
	_intRet: INT; // Return string converted to an integer
	_bResult : BOOL; // Output of the method
END_VAR
_inst_intStep := intGetPressureStep;
bGetPressureBusy := TRUE;

_bResult := FALSE;
CASE _inst_intStep OF
	0: // Wait for no error and router not busy
		IF NOT THIS^.P_bError AND NOT bRouterBusy THEN
			bRouterBusy := TRUE;
			_inst_intStep := _inst_intStep + 10;
		END_IF
		
	10: // Initialize parameters
		THIS^.M_LogMessage(_strSTART_MSG);
		_inst_fbParams.M_ClearParameters();
		// ADD ANY PARAMETERS HERE
		_inst_fbParams.M_OutputToParameterList(_inst_arrParams);
		_inst_intStep := _inst_intStep + 10;
		
	20: // Route the command
		_bComplete := M_RouterHelper(
			_in_strMethodName := _strCOMMAND_NAME, 
			_in_timeTimeout := _timeCOMMAND_TIMEOUT,
			_inout_arrParams := _inst_arrParams,
			_inout_arrOutputs := _inst_arrOutputs,
			_out_strReturnValue=>_inst_strRet);
		
		// If route completed, move to next step
		IF _bComplete THEN
			_inst_intStep := _inst_intStep + 10;
			bRouterBusy := FALSE;
		ELSIF THIS^.P_bError THEN
			_inst_intStep := 0;
			bRouterBusy := FALSE;
		END_IF
		
	30: // Parse results
		_intRet := STRING_TO_INT(_inst_strRet);
		IF _intRet > 0 THEN
			_bResult := TRUE;
			THIS^.M_LogMessage(_strEND_MSG);
			// DO ANY PARSING HERE
			_out_lrealPressure := _inst_fbParams.M_ParseDouble(_inst_fbParams.M_GetParameter('Pressure'));
//			_inst_fbParams.M_LoadFromParameterList(_inst_arrOutputs);
//			bEnabled := _inst_fbParams.M_ParseBool(_inst_fbParams.M_GetParameter('enabled'));
//			THIS^.bEnabled := bEnabled;			
			
		// Set error if command failed
		ELSE
			THIS^.M_SetError(_udintERROR_ID, _strERROR_MSG);
		END_IF
		
		// Go back to start
		_inst_intStep := 0;
END_CASE
M_GetPressure := _bResult;
intGetPressureStep := _inst_intStep;
END_METHOD

ACTION A_CommandRecovery:
IF NOT bGetPressureBusy AND intGetPressureStep > 0 THEN
	intGetPressureStep := 0;
	bRouterBusy := FALSE;
	THIS^.M_LogWarning('Get Pressure ended prematurely!');
END_IF
bGetPressureBusy := FALSE;

IF NOT bConnectBusy AND intConnectStep > 0 THEN
	intConnectStep := 0;
	bRouterBusy := FALSE;
	THIS^.M_LogWarning('Connect ended prematurely!');
END_IF
bConnectBusy := FALSE;

IF NOT bDisconnectBusy AND intDisconnectStep > 0 THEN
	intDisconnectStep := 0;
	bRouterBusy := FALSE;
	THIS^.M_LogWarning('Disconnect ended prematurely!');
END_IF
bDisconnectBusy := FALSE;

IF NOT bGetAlicatAbsDataBusy AND intGetAlicatAbsDataStep > 0 THEN
	intGetAlicatAbsDataStep := 0;
	bRouterBusy := FALSE;
	THIS^.M_LogWarning('GetAlicatAbsData ended prematurely!');
END_IF
bGetAlicatAbsDataBusy := FALSE;

IF NOT bLockDisplayBusy AND intLockDisplayStep > 0 THEN
	intLockDisplayStep := 0;
	bRouterBusy := FALSE;
	THIS^.M_LogWarning('LockDisplay ended prematurely!');
END_IF
bLockDisplayBusy := FALSE;

IF NOT bUnlockDisplayBusy AND intUnlockDisplayStep > 0 THEN
	intUnlockDisplayStep := 0;
	bRouterBusy := FALSE;
	THIS^.M_LogWarning('UnlockDisplay ended prematurely!');
END_IF
bUnlockDisplayBusy := FALSE;

IF NOT bTareBusy AND intTareStep > 0 THEN
	intTareStep := 0;
	bRouterBusy := FALSE;
	THIS^.M_LogWarning('Tare ended prematurely!');
END_IF
bTareBusy := FALSE;

IF NOT bRouterHelperBusy AND intRouterHelperStep > 0 THEN
	intRouterHelperStep := 0;
	THIS^.M_LogWarning('Router helper ended prematurely!');
END_IF
bRouterHelperBusy := FALSE;
END_ACTION

(*
Sends the given method to the API and receives and partially parses the result.
*)
METHOD PRIVATE M_RouterHelper : BOOL
VAR_INPUT
	(* Name of the method to call. *)
	_in_strMethodName : T_MaxString;
	(* Maximum time to wait for method response. *)
	_in_timeTimeout : TIME;
END_VAR
VAR_IN_OUT
	(* The array of parameters to send to the API. *)
	_inout_arrParams : T_ApiParameterList;
	(* The array that gets populated with any method output data. *)
	_inout_arrOutputs : T_ApiParameterList;
END_VAR
VAR_OUTPUT
	(* JSON string of the method return value. *)
	_out_strReturnValue: T_ApiParamValue;
END_VAR
VAR_INST
	(* Current step. *)
	_inst_intStep: INT;
	(* True if the method executed. *)
	_inst_bExec: BOOL;
	(* Return string of the method. *)
	_inst_strRet: T_ApiParamValue;
END_VAR
VAR
	(* True once the command routing finishes. *)
	_bComplete: BOOL;
	(* True once the API connects. *)
	_bApiConnect: BOOL;
END_VAR
_inst_intStep := intRouterHelperStep;
bRouterHelperBusy := TRUE;

CASE _inst_intStep OF
	0: // Start process only if there is no error on this FB
		IF NOT THIS^.P_bError THEN
			_inst_intStep := 10;
		END_IF
		
	10: // Check if command router connected
		IF NOT in_fbApi.P_bConnected THEN
			_inst_intStep := 20; // Go to API connect step
		ELSE
			_inst_intStep := 30; // Go to route command step
		END_IF
		
	20: // Connect the command router
		_bApiConnect := in_fbApi.M_Connect();
		IF _bApiConnect THEN
			_inst_intStep := _inst_intStep + 10; // Go to next step
		ELSIF in_fbApi.P_bError THEN
			THIS^.M_SetError(E_Alicat_Error.CommandRouterError, 'Error on command router function block while connecting!');
			_inst_intStep := 0; // Go back to start
		END_IF
		
	30:	// Route the command
		_bComplete := in_fbApi.M_RouteCommand(
			_in_strModuleId := in_strUniqueId,
			_in_strMethodName := _in_strMethodName,
			_in_timeTimeout := _in_timeTimeout,
			_inout_arrParameters := _inout_arrParams,
			_inout_arrOutputs := _inout_arrOutputs,
			_out_bCommandExecuted => _inst_bExec,
			_out_strReturnValue => _inst_strRet);
		IF _bComplete THEN
			_inst_intStep := _inst_intStep + 10; // Go to next step
		ELSIF in_fbApi.P_bError THEN
			THIS^.M_SetError(E_Alicat_Error.CommandRouterError, 'Error on command router function block while routing command!');
			_inst_intStep := 0; // Go back to start
		END_IF
		
	40: // Check result then go back to start
		IF NOT _inst_bExec THEN
			THIS^.M_SetError(E_Alicat_Error.CommandFault, 'Method in API failed to execute!');
		ELSE
			_out_strReturnValue := _inst_strRet;
			M_RouterHelper := TRUE;
		END_IF
		_inst_intStep := 0; // Go back to start
END_CASE
intRouterHelperStep := _inst_intStep;
END_METHOD

END_FUNCTION_BLOCK

// Concrete/Alicat/AlicatDifferential/FB_AlicatDifferential
FUNCTION_BLOCK FB_AlicatDifferential EXTENDS FB_PressureTransducer IMPLEMENTS I_PressureSensing, I_Connectable, I_DeviceInfo
VAR_INPUT
	in_fbApi : REFERENCE TO FB_CommandRouter;
END_VAR
VAR_OUTPUT
END_VAR
VAR
	//Copied all the variables from UReSeries program - still not sure which all we need
	bConnected: BOOL; // Value of P_bConnected
	bEnabled: BOOL; // Value of P_bEnabled
	bPoweredOn: BOOL; // Value of P_bPoweredOn
	strLoadedProgram: STRING(255); // Value of P_strLoadedProgram
	enumProgramState: E_PROGRAMSTATE; // Value of P_enumProgramState
	bRouterBusy: BOOL; // TRUE while M_RouterHelper is being used by a method
	bResetBusy: BOOL; // Value of P_bResetBusy
	//ST Adding parameters below
	bDisconnected: BOOL;
	bGetPressureSuccessful: BOOL;
	bGetAlicatDataSuccessful: BOOL;
	bLockDisplaySuccessful: BOOL;
	bUnlockDisplaySuccessful: BOOL;
	
	//Command Steps
	intGetPressureStep		 : INT;
	intConnectStep	  		 : INT;
	intDisconnectStep 		 : INT;
	intGetAlicatDiffDataStep : INT;
	intLockDisplayStep		 : INT;
	intUnlockDisplayStep	 : INT;
	intTareStep			  	 : INT;
	intRouterHelperStep	     : INT;
	
	
	//CommandBusy Bits
	bGetPressureBusy 	   : BOOL;
	bConnectBusy	 	   : BOOL;
	bDisconnectBusy  	   : BOOL;
	bGetAlicatDiffDataBusy : BOOL;
	bLockDisplayBusy	   : BOOL;
	bUnlockDisplayBusy	   : BOOL;
	bTareBusy			   : BOOL;
	bRouterHelperBusy	   : BOOL;
	
END_VAR

A_CommandRecovery();

(* This method returns the Pressure Value from the Alicat Differential Pressure Gauge.
Once the Pressure value is obtained, this method must return TRUE*)
METHOD M_GetAlicatDiffData : BOOL
VAR_INPUT
END_VAR
VAR_OUTPUT
	(*_output/input_datatypeName*)
	_out_lrealPressure	: LREAL;
	_out_stResult : ST_SerialDataFrame;
END_VAR
VAR CONSTANT
	_strCOMMAND_NAME : T_MaxString	:= 'GetAlicatDiffData'; // Name of the API method
	_timeCOMMAND_TIMEOUT : TIME		:= T#5S; // Max time to receive API response
	_strSTART_MSG : T_MaxString		:= 'Reading Alicat Serial Frame'; // Prints when method starts
	_strEND_MSG : T_MaxString		:= 'Read Alicat Serial Frame successfully'; // Prints when method finishes
	_udintERROR_ID : UDINT			:= E_Alicat_Error.FailedToReadSerialData; // Error ID to set if command fails
	_strERROR_MSG : T_MaxString		:= 'Failed to read Alicat Serial Frame!'; // Error message to set if command fails
END_VAR
VAR_INST
	_inst_arrParams: T_ApiParameterList; // Parameters array
	_inst_arrOutputs: T_ApiParameterList; // Outputs array
	_inst_strRet: T_ApiParamValue; // Return string from the router
	_inst_intStep: INT; // Current method step
	_inst_fbParams: FB_ApiParamBuilder; // Parameter builder FB
END_VAR
VAR
	_bComplete: BOOL; // True if the routing finishes
	_intRet: INT; // Return string converted to an integer
	_bResult : BOOL; // Output of the method
	_pStructPointer : PVOID; // Pointer to the struct
	_pStructPointerDiff : PVOID; 
END_VAR
_inst_intStep := intGetAlicatDiffDataStep;
bGetAlicatDiffDataBusy := TRUE;

_bResult := FALSE;
CASE _inst_intStep OF
	0: // Wait for no error and router not busy
		IF NOT THIS^.P_bError AND NOT bRouterBusy THEN
			bRouterBusy := TRUE;
			_inst_intStep := _inst_intStep + 10;
		END_IF
		
	10: // Initialize parameters
		THIS^.M_LogMessage(_strSTART_MSG);
		_inst_fbParams.M_ClearParameters();
		// ADD ANY PARAMETERS HERE
		_inst_fbParams.M_OutputToParameterList(_inst_arrParams);
		_inst_intStep := _inst_intStep + 10;
		
	20: // Route the command
		_bComplete := M_RouterHelper(
			_in_strMethodName := _strCOMMAND_NAME, 
			_in_timeTimeout := _timeCOMMAND_TIMEOUT,
			_inout_arrParams := _inst_arrParams,
			_inout_arrOutputs := _inst_arrOutputs,
			_out_strReturnValue=>_inst_strRet);
		
		// If route completed, move to next step
		IF _bComplete THEN
			_inst_intStep := _inst_intStep + 10;
			bRouterBusy := FALSE;
		ELSIF THIS^.P_bError THEN
			_inst_intStep := 0;
			bRouterBusy := FALSE;
		END_IF
		
	30: // Parse results
		_intRet := STRING_TO_INT(_inst_strRet);
		IF _intRet > 0 THEN
			_bResult := TRUE;
			THIS^.M_LogMessage(_strEND_MSG);
			// DO ANY PARSING HERE
			_pStructPointer := _inst_fbParams.M_GetParameter('alicatDiffDataFrame');	//Because this is the name of the parameter on the API side - type doesn't matter?
			
			_pStructPointerDiff := _inst_fbParams.M_GetStructMember(_pStructPointer, 'AlicatDifferentialDataFrame');	//Because AlicatDifferentialDataFrame is a member of the main struct on the API side			
		
			_out_stResult.stAlicatDiff.strDeviceID := _inst_fbParams.M_ParseString(_inst_fbParams.M_GetStructMember(_pStructPointerDiff, 'DeviceID'));
			_out_stResult.stAlicatDiff.lrDiffPressure := _inst_fbParams.M_ParseDouble(_inst_fbParams.M_GetStructMember(_pStructPointerDiff, 'DiffPressure'));
			_out_stResult.stAlicatDiff.strStatusCode := _inst_fbParams.M_ParseString(_inst_fbParams.M_GetStructMember(_pStructPointerDiff, 'StatusCode'));
			
			_out_lrealPressure := _out_stResult.stAlicatDiff.lrDiffPressure;
			
//			_inst_fbParams.M_LoadFromParameterList(_inst_arrOutputs);
//			bConnected := _inst_fbParams.M_ParseBool(_inst_fbParams.M_GetParameter('connected'));
//			THIS^.bConnected := bConnected;
			
		// Set error if command failed
		ELSE
			THIS^.M_SetError(_udintERROR_ID, _strERROR_MSG);
		END_IF
		
		// Go back to start
		_inst_intStep := 0;
END_CASE
M_GetAlicatDiffData := _bResult;
intgetAlicatDiffDataStep := _inst_intStep;
END_METHOD

(* This method returns the status of whether the screen on the device has been locked.
Once the screen is locked, this method must return TRUE*)
METHOD M_LockDisplay : BOOL
VAR_INPUT
END_VAR
VAR CONSTANT
	_strCOMMAND_NAME : T_MaxString	:= 'LockDisplay'; // Name of the API method
	_timeCOMMAND_TIMEOUT : TIME		:= T#2S; // Max time to receive API response
	_strSTART_MSG : T_MaxString		:= 'Locking Alicat Display'; // Prints when method starts
	_strEND_MSG : T_MaxString		:= 'Locked Alicat Display'; // Prints when method finishes
	_udintERROR_ID : UDINT			:= E_Alicat_Error.FailedToLockDisplay; // Error ID to set if command fails
	_strERROR_MSG : T_MaxString		:= 'Failed to lock display!'; // Error message to set if command fails
END_VAR
VAR_INST
	_inst_arrParams: T_ApiParameterList; // Parameters array
	_inst_arrOutputs: T_ApiParameterList; // Outputs array
	_inst_strRet: T_ApiParamValue; // Return string from the router
	_inst_intStep: INT; // Current method step
	_inst_fbParams: FB_ApiParamBuilder; // Parameter builder FB
END_VAR
VAR
	_bComplete: BOOL; // True if the routing finishes
	_intRet: INT; // Return string converted to an integer
	_bResult : BOOL; // Output of the method
END_VAR
_inst_intStep := intLockDisplayStep;
bLockDisplayBusy := TRUE;

_bResult := FALSE;
CASE _inst_intStep OF
	0: // Wait for no error and router not busy
		IF NOT THIS^.P_bError AND NOT bRouterBusy THEN
			bRouterBusy := TRUE;
			_inst_intStep := _inst_intStep + 10;
		END_IF
		
	10: // Initialize parameters
		THIS^.M_LogMessage(_strSTART_MSG);
		_inst_fbParams.M_ClearParameters();
		// ADD ANY PARAMETERS HERE
		_inst_fbParams.M_OutputToParameterList(_inst_arrParams);
		_inst_intStep := _inst_intStep + 10;
		
	20: // Route the command
		_bComplete := M_RouterHelper(
			_in_strMethodName := _strCOMMAND_NAME, 
			_in_timeTimeout := _timeCOMMAND_TIMEOUT,
			_inout_arrParams := _inst_arrParams,
			_inout_arrOutputs := _inst_arrOutputs,
			_out_strReturnValue=>_inst_strRet);
		
		// If route completed, move to next step
		IF _bComplete THEN
			_inst_intStep := _inst_intStep + 10;
			bRouterBusy := FALSE;
		ELSIF THIS^.P_bError THEN
			_inst_intStep := 0;
			bRouterBusy := FALSE;
		END_IF
		
	30: // Parse results
		_intRet := STRING_TO_INT(_inst_strRet);
		IF _intRet > 0 THEN
			_bResult := TRUE;
			THIS^.M_LogMessage(_strEND_MSG);
			// DO ANY PARSING HERE
//			_inst_fbParams.M_LoadFromParameterList(_inst_arrOutputs);
//			bConnected := _inst_fbParams.M_ParseBool(_inst_fbParams.M_GetParameter('connected'));
//			THIS^.bConnected := bConnected;
			
		// Set error if command failed
		ELSE
			THIS^.M_SetError(_udintERROR_ID, _strERROR_MSG);
		END_IF
		
		// Go back to start
		_inst_intStep := 0;
END_CASE
M_LockDisplay := _bResult;
intLockDisplayStep := _inst_intStep;
END_METHOD

(*This method returns whether the gauge pressure has been tared in the Differential Pressure Transducer.
Once the taring is complete, this method must return TRUE*)
METHOD M_Tare : BOOL
VAR_INPUT
END_VAR
VAR CONSTANT
	_strCOMMAND_NAME : T_MaxString	:= 'Tare'; // Name of the API method
	_timeCOMMAND_TIMEOUT : TIME		:= T#2S; // Max time to receive API response
	_strSTART_MSG : T_MaxString		:= 'Taring Gauge Pressure'; // Prints when method starts
	_strEND_MSG : T_MaxString		:= 'Tared Gauge Pressure'; // Prints when method finishes
	_udintERROR_ID : UDINT			:= E_Alicat_Error.FailedToTareDifferentialGauge; // Error ID to set if command fails
	_strERROR_MSG : T_MaxString		:= 'Failed to tare gauge!'; // Error message to set if command fails
END_VAR
VAR_INST
	_inst_arrParams: T_ApiParameterList; // Parameters array
	_inst_arrOutputs: T_ApiParameterList; // Outputs array
	_inst_strRet: T_ApiParamValue; // Return string from the router
	_inst_intStep: INT; // Current method step
	_inst_fbParams: FB_ApiParamBuilder; // Parameter builder FB
END_VAR
VAR
	_bComplete: BOOL; // True if the routing finishes
	_intRet: INT; // Return string converted to an integer
	_bResult : BOOL; // Output of the method
END_VAR
_inst_intStep := intTareStep;
bTareBusy	  := TRUE;

_bResult := FALSE;
CASE _inst_intStep OF
	0: // Wait for no error and router not busy
		IF NOT THIS^.P_bError AND NOT bRouterBusy THEN
			bRouterBusy := TRUE;
			_inst_intStep := _inst_intStep + 10;
		END_IF
		
	10: // Initialize parameters
		THIS^.M_LogMessage(_strSTART_MSG);
		_inst_fbParams.M_ClearParameters();
		// ADD ANY PARAMETERS HERE
		_inst_fbParams.M_OutputToParameterList(_inst_arrParams);
		_inst_intStep := _inst_intStep + 10;
		
	20: // Route the command
		_bComplete := M_RouterHelper(
			_in_strMethodName := _strCOMMAND_NAME, 
			_in_timeTimeout := _timeCOMMAND_TIMEOUT,
			_inout_arrParams := _inst_arrParams,
			_inout_arrOutputs := _inst_arrOutputs,
			_out_strReturnValue=>_inst_strRet);
		
		// If route completed, move to next step
		IF _bComplete THEN
			_inst_intStep := _inst_intStep + 10;
			bRouterBusy := FALSE;
		ELSIF THIS^.P_bError THEN
			_inst_intStep := 0;
			bRouterBusy := FALSE;
		END_IF
		
	30: // Parse results
		_intRet := STRING_TO_INT(_inst_strRet);
		IF _intRet > 0 THEN
			_bResult := TRUE;
			THIS^.M_LogMessage(_strEND_MSG);
			// DO ANY PARSING HERE
//			_inst_fbParams.M_LoadFromParameterList(_inst_arrOutputs);
//			bConnected := _inst_fbParams.M_ParseBool(_inst_fbParams.M_GetParameter('connected'));
//			THIS^.bConnected := bConnected;
			
		// Set error if command failed
		ELSE
			THIS^.M_SetError(_udintERROR_ID, _strERROR_MSG);
		END_IF
		
		// Go back to start
		_inst_intStep := 0;
END_CASE
M_Tare := _bResult;
intTareStep := _inst_intStep;
END_METHOD

(* This method returns the status of whether the screen on the device has been locked.
Once the screen is locked, this method must return TRUE*)
METHOD M_UnlockDisplay : BOOL
VAR_INPUT
END_VAR
VAR CONSTANT
	_strCOMMAND_NAME : T_MaxString	:= 'UnlockDisplay'; // Name of the API method
	_timeCOMMAND_TIMEOUT : TIME		:= T#2S; // Max time to receive API response
	_strSTART_MSG : T_MaxString		:= 'Unlocking Alicat Display'; // Prints when method starts
	_strEND_MSG : T_MaxString		:= 'Unlocked Alicat Display'; // Prints when method finishes
	_udintERROR_ID : UDINT			:= E_Alicat_Error.FailedToUnlockDisplay; // Error ID to set if command fails
	_strERROR_MSG : T_MaxString		:= 'Failed to unlock display!'; // Error message to set if command fails
END_VAR
VAR_INST
	_inst_arrParams: T_ApiParameterList; // Parameters array
	_inst_arrOutputs: T_ApiParameterList; // Outputs array
	_inst_strRet: T_ApiParamValue; // Return string from the router
	_inst_intStep: INT; // Current method step
	_inst_fbParams: FB_ApiParamBuilder; // Parameter builder FB
END_VAR
VAR
	_bComplete: BOOL; // True if the routing finishes
	_intRet: INT; // Return string converted to an integer
	_bResult : BOOL; // Output of the method
END_VAR
_inst_intStep := intUnlockDisplayStep;
bUnlockDisplayBusy := TRUE;

_bResult := FALSE;
CASE _inst_intStep OF
	0: // Wait for no error and router not busy
		IF NOT THIS^.P_bError AND NOT bRouterBusy THEN
			bRouterBusy := TRUE;
			_inst_intStep := _inst_intStep + 10;
		END_IF
		
	10: // Initialize parameters
		THIS^.M_LogMessage(_strSTART_MSG);
		_inst_fbParams.M_ClearParameters();
		// ADD ANY PARAMETERS HERE
		_inst_fbParams.M_OutputToParameterList(_inst_arrParams);
		_inst_intStep := _inst_intStep + 10;
		
	20: // Route the command
		_bComplete := M_RouterHelper(
			_in_strMethodName := _strCOMMAND_NAME, 
			_in_timeTimeout := _timeCOMMAND_TIMEOUT,
			_inout_arrParams := _inst_arrParams,
			_inout_arrOutputs := _inst_arrOutputs,
			_out_strReturnValue=>_inst_strRet);
		
		// If route completed, move to next step
		IF _bComplete THEN
			_inst_intStep := _inst_intStep + 10;
			bRouterBusy := FALSE;
		ELSIF THIS^.P_bError THEN
			_inst_intStep := 0;
			bRouterBusy := FALSE;
		END_IF
		
	30: // Parse results
		_intRet := STRING_TO_INT(_inst_strRet);
		IF _intRet > 0 THEN
			_bResult := TRUE;
			THIS^.M_LogMessage(_strEND_MSG);
			// DO ANY PARSING HERE
//			_inst_fbParams.M_LoadFromParameterList(_inst_arrOutputs);
//			bConnected := _inst_fbParams.M_ParseBool(_inst_fbParams.M_GetParameter('connected'));
//			THIS^.bConnected := bConnected;
			
		// Set error if command failed
		ELSE
			THIS^.M_SetError(_udintERROR_ID, _strERROR_MSG);
		END_IF
		
		// Go back to start
		_inst_intStep := 0;
END_CASE
M_UnlockDisplay := _bResult;
intUnlockDisplayStep := _inst_intStep;
END_METHOD

(* This method should establish any external connections required to use the
	functions of the device, and return TRUE and set P_bConnected to TRUE once
	connected. *)
METHOD M_Connect : BOOL
VAR CONSTANT
	_strCOMMAND_NAME : T_MaxString	:= 'Connect'; // Name of the API method
	_timeCOMMAND_TIMEOUT : TIME		:= T#100S; // Max time to receive API response
	_strSTART_MSG : T_MaxString		:= 'Connecting'; // Prints when method starts
	_strEND_MSG : T_MaxString		:= 'Connected'; // Prints when method finishes
	_udintERROR_ID : UDINT			:= E_Alicat_Error.FailedToConnect; // Error ID to set if command fails
	_strERROR_MSG : T_MaxString		:= 'Failed to connect to Differential Pressure Transducer!'; // Error message to set if command fails
END_VAR
VAR_INST
	_inst_arrParams: T_ApiParameterList; // Parameters array
	_inst_arrOutputs: T_ApiParameterList; // Outputs array
	_inst_strRet: T_ApiParamValue; // Return string from the router
	_inst_intStep: INT; // Current method step
	_inst_fbParams: FB_ApiParamBuilder; // Parameter builder FB
END_VAR
VAR
	_bComplete: BOOL; // True if the routing finishes
	_intRet: INT; // Return string converted to an integer
	_bResult : BOOL; // Output of the method
END_VAR
_inst_intStep := intConnectStep;
bConnectBusy  := TRUE;

_bResult := FALSE;
CASE _inst_intStep OF
	0: // Wait for no error and router not busy
		IF NOT THIS^.P_bError AND NOT bRouterBusy THEN
			bRouterBusy := TRUE;
			_inst_intStep := _inst_intStep + 10;
		END_IF
		
	10: // Initialize parameters
		THIS^.M_LogMessage(_strSTART_MSG);
		_inst_fbParams.M_ClearParameters();
		// ADD ANY PARAMETERS HERE
		_inst_fbParams.M_OutputToParameterList(_inst_arrParams);
		_inst_intStep := _inst_intStep + 10;
		
	20: // Route the command
		_bComplete := M_RouterHelper(
			_in_strMethodName := _strCOMMAND_NAME, 
			_in_timeTimeout := _timeCOMMAND_TIMEOUT,
			_inout_arrParams := _inst_arrParams,
			_inout_arrOutputs := _inst_arrOutputs,
			_out_strReturnValue=>_inst_strRet);
		
		// If route completed, move to next step
		IF _bComplete THEN
			_inst_intStep := _inst_intStep + 10;
			bRouterBusy := FALSE;
		ELSIF THIS^.P_bError THEN
			_inst_intStep := 0;
			bRouterBusy := FALSE;
		END_IF
		
	30: // Parse results
		_intRet := STRING_TO_INT(_inst_strRet);
		IF _intRet > 0 THEN
			_bResult := TRUE;
			THIS^.M_LogMessage(_strEND_MSG);
			// DO ANY PARSING HERE
			bConnected := TRUE;
			
		// Set error if command failed
		ELSE
			THIS^.M_SetError(_udintERROR_ID, _strERROR_MSG);
		END_IF
		
		// Go back to start
		_inst_intStep := 0;
END_CASE
M_Connect := _bResult;
intConnectStep := _inst_intStep;
END_METHOD

(* This method should break any connections established by M_Connect. It should
	immediately set P_bConnected to false unless all connections are known to
	be still active, and return TRUE once those connections are all fully
	disconnected. *)
METHOD M_Disconnect : BOOL
VAR CONSTANT
	_strCOMMAND_NAME : T_MaxString	:= 'Disconnect'; // Name of the API method
	_timeCOMMAND_TIMEOUT : TIME		:= T#30S; // Max time to receive API response
	_strSTART_MSG : T_MaxString		:= 'Disconnecting'; // Prints when method starts
	_strEND_MSG : T_MaxString		:= 'Disconnected'; // Prints when method finishes
	_udintERROR_ID : UDINT			:= E_Alicat_Error.FailedToDisconnect; // Error ID to set if command fails
	_strERROR_MSG : T_MaxString		:= 'Failed to disconnect from Differential Pressure Transducer!'; // Error message to set if command fails
END_VAR
VAR_INST
	_inst_arrParams: T_ApiParameterList; // Parameters array
	_inst_arrOutputs: T_ApiParameterList; // Outputs array
	_inst_strRet: T_ApiParamValue; // Return string from the router
	_inst_intStep: INT; // Current method step
	_inst_fbParams: FB_ApiParamBuilder; // Parameter builder FB
END_VAR
VAR
	_bComplete: BOOL; // True if the routing finishes
	_intRet: INT; // Return string converted to an integer
	_bResult : BOOL; // Output of the method
END_VAR
_inst_intStep   := intDisconnectStep;
bDisconnectBusy := TRUE;

_bResult := FALSE;
CASE _inst_intStep OF
	0: // Wait for no error and router not busy
		IF NOT THIS^.P_bError AND NOT bRouterBusy THEN
			bRouterBusy := TRUE;
			_inst_intStep := _inst_intStep + 10;
		END_IF
		
	10: // Initialize parameters
		THIS^.M_LogMessage(_strSTART_MSG);
		_inst_fbParams.M_ClearParameters();
		// ADD ANY PARAMETERS HERE
		_inst_fbParams.M_OutputToParameterList(_inst_arrParams);
		_inst_intStep := _inst_intStep + 10;
		
	20: // Route the command
		_bComplete := M_RouterHelper(
			_in_strMethodName := _strCOMMAND_NAME, 
			_in_timeTimeout := _timeCOMMAND_TIMEOUT,
			_inout_arrParams := _inst_arrParams,
			_inout_arrOutputs := _inst_arrOutputs,
			_out_strReturnValue=>_inst_strRet);
		
		// If route completed, move to next step
		IF _bComplete THEN
			_inst_intStep := _inst_intStep + 10;
			bRouterBusy := FALSE;
		ELSIF THIS^.P_bError THEN
			_inst_intStep := 0;
			bRouterBusy := FALSE;
		END_IF
		
	30: // Parse results
		_intRet := STRING_TO_INT(_inst_strRet);
		IF _intRet > 0 THEN
			_bResult := TRUE;
			THIS^.M_LogMessage(_strEND_MSG);
			// DO ANY PARSING HERE
			bConnected := FALSE;
			
		// Set error if command failed
		ELSE
			THIS^.M_SetError(_udintERROR_ID, _strERROR_MSG);
		END_IF
		
		// Go back to start
		_inst_intStep := 0;
END_CASE
M_Disconnect := _bResult;
intDisconnectStep := _inst_intStep;
END_METHOD

(* This method should explicitly check the connection status of the device.
	Once the connection status is known, this method should return TRUE.
	If this method fails, P_bConnected should be set to FALSE since the device
	is not absolutely known to still be connected. *)
METHOD M_GetConnectStatus : BOOL
VAR_OUTPUT
	(* This should return TRUE if all connections required to make the device
		function properly are known to be connected, and FALSE otherwise. *)
	bConnected	: BOOL;
END_VAR
bConnected := P_bConnected;
M_GetConnectStatus := TRUE;
THIS^.M_LogWarning('Get connect status not implemented in FB_Differential!');
END_METHOD

(* This property should be TRUE while any method in this interface is actively
	executing, or FALSE otherwise. *)
PROPERTY P_bConnectBusy : BOOL
GET
END_GET
END_PROPERTY

(* This should be set to TRUE if M_Connect is successful or M_GetConnectStatus
	determines the device to be connected, and set to FALSE if M_Disconnect is
	called at all, M_GetConnectStatus fails, or M_GetConnectStatus determines
	the device to be not connected. *)
PROPERTY P_bConnected : BOOL
GET
END_GET
END_PROPERTY

PROPERTY P_strDescription : Sensata_Common.T_MaxString
GET
END_GET
END_PROPERTY

PROPERTY P_strMake : Sensata_Common.T_MaxString
GET
END_GET
END_PROPERTY

PROPERTY P_strModel : Sensata_Common.T_MaxString
GET
END_GET
END_PROPERTY

PROPERTY P_strVersion : Sensata_Common.T_MaxString
GET
END_GET
END_PROPERTY

(* This method returns the Pressure Value from the Alicat Differential Pressure Gauge.
Once the Pressure value is obtained, this method must return TRUE*)
METHOD M_GetPressure : BOOL
VAR_OUTPUT
	(*_output/input_datatypeName*)
	_out_lrealPressure	: LREAL;
END_VAR
VAR CONSTANT
	_strCOMMAND_NAME : T_MaxString	:= 'GetPressure'; // Name of the API method
	_timeCOMMAND_TIMEOUT : TIME		:= T#5S; // Max time to receive API response
	_strSTART_MSG : T_MaxString		:= 'Reading Pressure Value'; // Prints when method starts
	_strEND_MSG : T_MaxString		:= 'Pressure Read'; // Prints when method finishes
	_udintERROR_ID : UDINT			:= E_Alicat_Error.FailedToReadSerialData; // Error ID to set if command fails
	_strERROR_MSG : T_MaxString		:= 'Failed to read serial data and hence pressure!'; // Error message to set if command fails
END_VAR
VAR_INST
	_inst_arrParams: T_ApiParameterList; // Parameters array
	_inst_arrOutputs: T_ApiParameterList; // Outputs array
	_inst_strRet: T_ApiParamValue; // Return string from the router
	_inst_intStep: INT; // Current method step
	_inst_fbParams: FB_ApiParamBuilder; // Parameter builder FB
END_VAR
VAR
	_bComplete: BOOL; // True if the routing finishes
	_intRet: INT; // Return string converted to an integer
	_bResult : BOOL; // Output of the method
END_VAR
_inst_intStep := intGetPressureStep;
bConnectBusy  := TRUE;

_bResult := FALSE;
CASE _inst_intStep OF
	0: // Wait for no error and router not busy
		IF NOT THIS^.P_bError AND NOT bRouterBusy THEN
			bRouterBusy := TRUE;
			_inst_intStep := _inst_intStep + 10;
		END_IF
		
	10: // Initialize parameters
		THIS^.M_LogMessage(_strSTART_MSG);
		_inst_fbParams.M_ClearParameters();
		// ADD ANY PARAMETERS HERE
		_inst_fbParams.M_OutputToParameterList(_inst_arrParams);
		_inst_intStep := _inst_intStep + 10;
		
	20: // Route the command
		_bComplete := M_RouterHelper(
			_in_strMethodName := _strCOMMAND_NAME, 
			_in_timeTimeout := _timeCOMMAND_TIMEOUT,
			_inout_arrParams := _inst_arrParams,
			_inout_arrOutputs := _inst_arrOutputs,
			_out_strReturnValue=>_inst_strRet);
		
		// If route completed, move to next step
		IF _bComplete THEN
			_inst_intStep := _inst_intStep + 10;
			bRouterBusy := FALSE;
		ELSIF THIS^.P_bError THEN
			_inst_intStep := 0;
			bRouterBusy := FALSE;
		END_IF
		
	30: // Parse results
		_intRet := STRING_TO_INT(_inst_strRet);
		IF _intRet > 0 THEN
			_bResult := TRUE;
			THIS^.M_LogMessage(_strEND_MSG);
			// DO ANY PARSING HERE
			_out_lrealPressure := _inst_fbParams.M_ParseDouble(_inst_fbParams.M_GetParameter('Pressure'));
//			_inst_fbParams.M_LoadFromParameterList(_inst_arrOutputs);
//			bEnabled := _inst_fbParams.M_ParseBool(_inst_fbParams.M_GetParameter('enabled'));
//			THIS^.bEnabled := bEnabled;			
			
		// Set error if command failed
		ELSE
			THIS^.M_SetError(_udintERROR_ID, _strERROR_MSG);
		END_IF
		
		// Go back to start
		_inst_intStep := 0;
END_CASE
M_GetPressure := _bResult;
intGetPressureStep := _inst_intStep;
END_METHOD

ACTION A_CommandRecovery:
IF NOT bGetPressureBusy AND intGetPressureStep > 0 THEN
	intGetPressureStep := 0;
	bRouterBusy := FALSE;
	THIS^.M_LogWarning('Get Pressure ended prematurely!');
END_IF
bGetPressureBusy := FALSE;

IF NOT bConnectBusy AND intConnectStep > 0 THEN
	intConnectStep := 0;
	bRouterBusy := FALSE;
	THIS^.M_LogWarning('Connect ended prematurely!');
END_IF
bConnectBusy := FALSE;

IF NOT bDisconnectBusy AND intDisconnectStep > 0 THEN
	intDisconnectStep := 0;
	bRouterBusy := FALSE;
	THIS^.M_LogWarning('Disconnect ended prematurely!');
END_IF
bDisconnectBusy := FALSE;

IF NOT bGetAlicatDiffDataBusy AND intGetAlicatDiffDataStep > 0 THEN
	intGetAlicatDiffDataStep := 0;
	bRouterBusy := FALSE;
	THIS^.M_LogWarning('GetAlicatDiffData ended prematurely!');
END_IF
bGetAlicatDiffDataBusy := FALSE;

IF NOT bLockDisplayBusy AND intLockDisplayStep > 0 THEN
	intLockDisplayStep := 0;
	bRouterBusy := FALSE;
	THIS^.M_LogWarning('LockDisplay ended prematurely!');
END_IF
bLockDisplayBusy := FALSE;

IF NOT bUnlockDisplayBusy AND intUnlockDisplayStep > 0 THEN
	intUnlockDisplayStep := 0;
	bRouterBusy := FALSE;
	THIS^.M_LogWarning('UnlockDisplay ended prematurely!');
END_IF
bUnlockDisplayBusy := FALSE;

IF NOT bTareBusy AND intTareStep > 0 THEN
	intTareStep := 0;
	bRouterBusy := FALSE;
	THIS^.M_LogWarning('Tare ended prematurely!');
END_IF
bTareBusy := FALSE;

IF NOT bRouterHelperBusy AND intRouterHelperStep > 0 THEN
	intRouterHelperStep := 0;
	THIS^.M_LogWarning('Router helper ended prematurely!');
END_IF
bRouterHelperBusy := FALSE;
END_ACTION

(*
Sends the given method to the API and receives and partially parses the result.
*)
METHOD PRIVATE M_RouterHelper : BOOL
VAR_INPUT
	(* Name of the method to call. *)
	_in_strMethodName : T_MaxString;
	(* Maximum time to wait for method response. *)
	_in_timeTimeout : TIME;
END_VAR
VAR_IN_OUT
	(* The array of parameters to send to the API. *)
	_inout_arrParams : T_ApiParameterList;
	(* The array that gets populated with any method output data. *)
	_inout_arrOutputs : T_ApiParameterList;
END_VAR
VAR_OUTPUT
	(* JSON string of the method return value. *)
	_out_strReturnValue: T_ApiParamValue;
END_VAR
VAR_INST
	(* Current step. *)
	_inst_intStep: INT;
	(* True if the method executed. *)
	_inst_bExec: BOOL;
	(* Return string of the method. *)
	_inst_strRet: T_ApiParamValue;
END_VAR
VAR
	(* True once the command routing finishes. *)
	_bComplete: BOOL;
	(* True once the API connects. *)
	_bApiConnect: BOOL;
END_VAR
_inst_intStep := intRouterHelperStep;
bRouterHelperBusy := TRUE;

CASE _inst_intStep OF
	0: // Start process only if there is no error on this FB
		IF NOT THIS^.P_bError THEN
			_inst_intStep := 10;
		END_IF
		
	10: // Check if command router connected
		IF NOT in_fbApi.P_bConnected THEN
			_inst_intStep := 20; // Go to API connect step
		ELSE
			_inst_intStep := 30; // Go to route command step
		END_IF
		
	20: // Connect the command router
		_bApiConnect := in_fbApi.M_Connect();
		IF _bApiConnect THEN
			_inst_intStep := _inst_intStep + 10; // Go to next step
		ELSIF in_fbApi.P_bError THEN
			THIS^.M_SetError(E_Alicat_Error.CommandRouterError, 'Error on command router function block while connecting!');
			_inst_intStep := 0; // Go back to start
		END_IF
		
	30:	// Route the command
		_bComplete := in_fbApi.M_RouteCommand(
			_in_strModuleId := in_strUniqueId,
			_in_strMethodName := _in_strMethodName,
			_in_timeTimeout := _in_timeTimeout,
			_inout_arrParameters := _inout_arrParams,
			_inout_arrOutputs := _inout_arrOutputs,
			_out_bCommandExecuted => _inst_bExec,
			_out_strReturnValue => _inst_strRet);
		IF _bComplete THEN
			_inst_intStep := _inst_intStep + 10; // Go to next step
		ELSIF in_fbApi.P_bError THEN
			THIS^.M_SetError(E_Alicat_Error.CommandRouterError, 'Error on command router function block while routing command!');
			_inst_intStep := 0; // Go back to start
		END_IF
		
	40: // Check result then go back to start
		IF NOT _inst_bExec THEN
			THIS^.M_SetError(E_Alicat_Error.CommandFault, 'Method in API failed to execute!');
		ELSE
			_out_strReturnValue := _inst_strRet;
			M_RouterHelper := TRUE;
		END_IF
		_inst_intStep := 0; // Go back to start
END_CASE

intRouterHelperStep := _inst_intStep;
END_METHOD

END_FUNCTION_BLOCK

// Concrete/Alicat/AlicatFlowMeter/FB_AlicatFlowMeter
FUNCTION_BLOCK FB_AlicatFlowMeter EXTENDS FB_PressureTransducer IMPLEMENTS I_PressureSensing, I_Connectable, I_DeviceInfo
VAR_INPUT
	in_fbApi : REFERENCE TO FB_CommandRouter;
END_VAR
VAR_OUTPUT
END_VAR
VAR
	//Copied all the variables from UReSeries program - still not sure which all we need
	bConnected: BOOL; // Value of P_bConnected
	bEnabled: BOOL; // Value of P_bEnabled
	bPoweredOn: BOOL; // Value of P_bPoweredOn
	strLoadedProgram: STRING(255); // Value of P_strLoadedProgram
	enumProgramState: E_PROGRAMSTATE; // Value of P_enumProgramState
	bRouterBusy: BOOL; // TRUE while M_RouterHelper is being used by a method
	bResetBusy: BOOL; // Value of P_bResetBusy
	//ST Adding parameters below
	bDisconnected: BOOL;
	bGetPressureSuccessful: BOOL;
	bGetAlicatDataSuccessful: BOOL;
	bLockDisplaySuccessful: BOOL;
	bUnlockDisplaySuccessful: BOOL;
	
	//Command Steps
	intGetPressureStep		 : INT;
	intConnectStep	  		 : INT;
	intDisconnectStep 		 : INT;
	intGetAlicatFlowDataStep : INT;
	intLockDisplayStep		 : INT;
	intUnlockDisplayStep	 : INT;
	intTareStep			  	 : INT;
	intRouterHelperStep		 : INT;
	
	
	//CommandBusy Bits
	bGetPressureBusy 	   : BOOL;
	bConnectBusy	 	   : BOOL;
	bDisconnectBusy  	   : BOOL;
	bGetAlicatFlowDataBusy : BOOL;
	bLockDisplayBusy	   : BOOL;
	bUnlockDisplayBusy	   : BOOL;
	bTareBusy			   : BOOL;
	bRouterHelperBusy	   : BOOL;
	
END_VAR

A_CommandRecovery();

(* This method returns the Pressure Value from the Alicat Flow Meter.
Once the Pressure value is obtained, this method must return TRUE*)
METHOD M_GetAlicatFlowData : BOOL
VAR_INPUT
END_VAR
VAR_OUTPUT
	(*_output/input_datatypeName*)
	_out_lrealPressure	   : LREAL;
	_out_lrealTotFlow      : LREAL;
	_out_lrealMassFlowRate : LREAL;
	_out_lrealVolFlowRate  : LREAL;
	_out_stResult : ST_SerialDataFrame;
END_VAR
VAR CONSTANT
	_strCOMMAND_NAME : T_MaxString	:= 'GetAlicatFlowData'; // Name of the API method
	_timeCOMMAND_TIMEOUT : TIME		:= T#5S; // Max time to receive API response
	_strSTART_MSG : T_MaxString		:= 'Reading Alicat Serial Frame'; // Prints when method starts
	_strEND_MSG : T_MaxString		:= 'Read Alicat Serial Frame successfully'; // Prints when method finishes
	_udintERROR_ID : UDINT			:= E_Alicat_Error.FailedToReadSerialData; // Error ID to set if command fails
	_strERROR_MSG : T_MaxString		:= 'Failed to read Alicat Serial Frame!'; // Error message to set if command fails
END_VAR
VAR_INST
	_inst_arrParams: T_ApiParameterList; // Parameters array
	_inst_arrOutputs: T_ApiParameterList; // Outputs array
	_inst_strRet: T_ApiParamValue; // Return string from the router
	_inst_intStep: INT; // Current method step
	_inst_fbParams: FB_ApiParamBuilder; // Parameter builder FB
END_VAR
VAR
	_bComplete: BOOL; // True if the routing finishes
	_intRet: INT; // Return string converted to an integer
	_bResult : BOOL; // Output of the method
	_pStructPointer : PVOID; // Pointer to the struct
	_pStructPointerDiff : PVOID; 
END_VAR
_inst_intStep 		   := intGetAlicatFlowDataStep;
bGetAlicatFlowDataBusy := TRUE;


_bResult := FALSE;
CASE _inst_intStep OF
	0: // Wait for no error and router not busy
		IF NOT THIS^.P_bError AND NOT bRouterBusy THEN
			bRouterBusy := TRUE;
			_inst_intStep := _inst_intStep + 10;
		END_IF
		
	10: // Initialize parameters
		THIS^.M_LogMessage(_strSTART_MSG);
		_inst_fbParams.M_ClearParameters();
		// ADD ANY PARAMETERS HERE
		_inst_fbParams.M_OutputToParameterList(_inst_arrParams);
		_inst_intStep := _inst_intStep + 10;
		
	20: // Route the command
		_bComplete := M_RouterHelper(
			_in_strMethodName := _strCOMMAND_NAME, 
			_in_timeTimeout := _timeCOMMAND_TIMEOUT,
			_inout_arrParams := _inst_arrParams,
			_inout_arrOutputs := _inst_arrOutputs,
			_out_strReturnValue=>_inst_strRet);
		
		// If route completed, move to next step
		IF _bComplete THEN
			_inst_intStep := _inst_intStep + 10;
			bRouterBusy := FALSE;
		ELSIF THIS^.P_bError THEN
			_inst_intStep := 0;
			bRouterBusy := FALSE;
		END_IF
		
	30: // Parse results
		_intRet := STRING_TO_INT(_inst_strRet);
		IF _intRet > 0 THEN
			_bResult := TRUE;
			THIS^.M_LogMessage(_strEND_MSG);
			// DO ANY PARSING HERE
			_pStructPointer := _inst_fbParams.M_GetParameter('alicatFlowMeterDataFrame');	//Because this is the name of the parameter on the API side - type doesn't matter?
			
			_pStructPointerDiff := _inst_fbParams.M_GetStructMember(_pStructPointer, 'AlicatFlowMeter');	//Because AlicatAbsoluteDataFrame is a member of the main struct			
		
			_out_stResult.stAlicatFlow.strDeviceID := _inst_fbParams.M_ParseString(_inst_fbParams.M_GetStructMember(_pStructPointerDiff, 'DeviceID'));
			_out_stResult.stAlicatFlow.lrAbsPressure := _inst_fbParams.M_ParseDouble(_inst_fbParams.M_GetStructMember(_pStructPointerDiff, 'AbsPressure'));
			_out_stResult.stAlicatFlow.lrTemperature := _inst_fbParams.M_ParseDouble(_inst_fbParams.M_GetStructMember(_pStructPointerDiff, 'Temperature'));
			_out_stResult.stAlicatFlow.lrVolFlowRate := _inst_fbParams.M_ParseDouble(_inst_fbParams.M_GetStructMember(_pStructPointerDiff, 'VolumetricFlowRate'));
			_out_stResult.stAlicatFlow.lrMassFlowRate := _inst_fbParams.M_ParseDouble(_inst_fbParams.M_GetStructMember(_pStructPointerDiff, 'MassFlowRate'));
			_out_stResult.stAlicatFlow.lrTotalizedFlow := _inst_fbParams.M_ParseDouble(_inst_fbParams.M_GetStructMember(_pStructPointerDiff, 'TotalizedFlow'));
			_out_stResult.stAlicatFlow.strGasSelect := _inst_fbParams.M_ParseString(_inst_fbParams.M_GetStructMember(_pStructPointerDiff, 'GasSelect'));
			_out_stResult.stAlicatFlow.strStatusCode := _inst_fbParams.M_ParseString(_inst_fbParams.M_GetStructMember(_pStructPointerDiff, 'StatusCode'));
			
			_out_lrealPressure := _out_stResult.stAlicatFlow.lrAbsPressure;
			_out_lrealTotFlow  := _out_stResult.stAlicatFlow.lrTotalizedFlow;
			_out_lrealMassFlowRate := _out_stResult.stAlicatFlow.lrMassFlowRate;
			_out_lrealVolFlowRate := _out_stResult.stAlicatFlow.lrVolFlowRate;
			
//			_inst_fbParams.M_LoadFromParameterList(_inst_arrOutputs);
//			bConnected := _inst_fbParams.M_ParseBool(_inst_fbParams.M_GetParameter('connected'));
//			THIS^.bConnected := bConnected;
			
		// Set error if command failed
		ELSE
			THIS^.M_SetError(_udintERROR_ID, _strERROR_MSG);
		END_IF
		
		// Go back to start
		_inst_intStep := 0;
END_CASE
M_GetAlicatFlowData := _bResult;
intGetAlicatFlowDataStep := _inst_intStep;
END_METHOD

(* This method returns the status of whether the screen on the device has been locked.
Once the screen is locked, this method must return TRUE*)
METHOD M_LockDisplay : BOOL
VAR_INPUT
END_VAR
VAR CONSTANT
	_strCOMMAND_NAME : T_MaxString	:= 'LockDisplay'; // Name of the API method
	_timeCOMMAND_TIMEOUT : TIME		:= T#2S; // Max time to receive API response
	_strSTART_MSG : T_MaxString		:= 'Locking Alicat Display'; // Prints when method starts
	_strEND_MSG : T_MaxString		:= 'Locked Alicat Display'; // Prints when method finishes
	_udintERROR_ID : UDINT			:= E_Alicat_Error.FailedToLockDisplay; // Error ID to set if command fails
	_strERROR_MSG : T_MaxString		:= 'Failed to lock display!'; // Error message to set if command fails
END_VAR
VAR_INST
	_inst_arrParams: T_ApiParameterList; // Parameters array
	_inst_arrOutputs: T_ApiParameterList; // Outputs array
	_inst_strRet: T_ApiParamValue; // Return string from the router
	_inst_intStep: INT; // Current method step
	_inst_fbParams: FB_ApiParamBuilder; // Parameter builder FB
END_VAR
VAR
	_bComplete: BOOL; // True if the routing finishes
	_intRet: INT; // Return string converted to an integer
	_bResult : BOOL; // Output of the method
END_VAR
_inst_intStep    := intLockDisplayStep;
bLockDisplaybusy := TRUE;


_bResult := FALSE;
CASE _inst_intStep OF
	0: // Wait for no error and router not busy
		IF NOT THIS^.P_bError AND NOT bRouterBusy THEN
			bRouterBusy := TRUE;
			_inst_intStep := _inst_intStep + 10;
		END_IF
		
	10: // Initialize parameters
		THIS^.M_LogMessage(_strSTART_MSG);
		_inst_fbParams.M_ClearParameters();
		// ADD ANY PARAMETERS HERE
		_inst_fbParams.M_OutputToParameterList(_inst_arrParams);
		_inst_intStep := _inst_intStep + 10;
		
	20: // Route the command
		_bComplete := M_RouterHelper(
			_in_strMethodName := _strCOMMAND_NAME, 
			_in_timeTimeout := _timeCOMMAND_TIMEOUT,
			_inout_arrParams := _inst_arrParams,
			_inout_arrOutputs := _inst_arrOutputs,
			_out_strReturnValue=>_inst_strRet);
		
		// If route completed, move to next step
		IF _bComplete THEN
			_inst_intStep := _inst_intStep + 10;
			bRouterBusy := FALSE;
		ELSIF THIS^.P_bError THEN
			_inst_intStep := 0;
			bRouterBusy := FALSE;
		END_IF
		
	30: // Parse results
		_intRet := STRING_TO_INT(_inst_strRet);
		IF _intRet > 0 THEN
			_bResult := TRUE;
			THIS^.M_LogMessage(_strEND_MSG);
			// DO ANY PARSING HERE
//			_inst_fbParams.M_LoadFromParameterList(_inst_arrOutputs);
//			bConnected := _inst_fbParams.M_ParseBool(_inst_fbParams.M_GetParameter('connected'));
//			THIS^.bConnected := bConnected;
			
		// Set error if command failed
		ELSE
			THIS^.M_SetError(_udintERROR_ID, _strERROR_MSG);
		END_IF
		
		// Go back to start
		_inst_intStep := 0;
END_CASE
M_LockDisplay := _bResult;
intLockDisplayStep := _inst_intStep;
END_METHOD

(*This method returns whether the flow rate has been tared in the Alicat Flow Meter.
Once the taring is complete, this method must return TRUE*)
METHOD M_Tare : BOOL
VAR_INPUT
END_VAR
VAR CONSTANT
	_strCOMMAND_NAME : T_MaxString	:= 'Tare'; // Name of the API method
	_timeCOMMAND_TIMEOUT : TIME		:= T#2S; // Max time to receive API response
	_strSTART_MSG : T_MaxString		:= 'Taring Flow Rate'; // Prints when method starts
	_strEND_MSG : T_MaxString		:= 'Tared Flow Rate'; // Prints when method finishes
	_udintERROR_ID : UDINT			:= E_Alicat_Error.FailedToTareFlowMeter; // Error ID to set if command fails
	_strERROR_MSG : T_MaxString		:= 'Failed to tare flow rate!'; // Error message to set if command fails
END_VAR
VAR_INST
	_inst_arrParams: T_ApiParameterList; // Parameters array
	_inst_arrOutputs: T_ApiParameterList; // Outputs array
	_inst_strRet: T_ApiParamValue; // Return string from the router
	_inst_intStep: INT; // Current method step
	_inst_fbParams: FB_ApiParamBuilder; // Parameter builder FB
END_VAR
VAR
	_bComplete: BOOL; // True if the routing finishes
	_intRet: INT; // Return string converted to an integer
	_bResult : BOOL; // Output of the method
END_VAR
_inst_intStep := intTareStep;
bTareBusy	  := TRUE;

_bResult := FALSE;
CASE _inst_intStep OF
	0: // Wait for no error and router not busy
		IF NOT THIS^.P_bError AND NOT bRouterBusy THEN
			bRouterBusy := TRUE;
			_inst_intStep := _inst_intStep + 10;
		END_IF
		
	10: // Initialize parameters
		THIS^.M_LogMessage(_strSTART_MSG);
		_inst_fbParams.M_ClearParameters();
		// ADD ANY PARAMETERS HERE
		_inst_fbParams.M_OutputToParameterList(_inst_arrParams);
		_inst_intStep := _inst_intStep + 10;
		
	20: // Route the command
		_bComplete := M_RouterHelper(
			_in_strMethodName := _strCOMMAND_NAME, 
			_in_timeTimeout := _timeCOMMAND_TIMEOUT,
			_inout_arrParams := _inst_arrParams,
			_inout_arrOutputs := _inst_arrOutputs,
			_out_strReturnValue=>_inst_strRet);
		
		// If route completed, move to next step
		IF _bComplete THEN
			_inst_intStep := _inst_intStep + 10;
			bRouterBusy := FALSE;
		ELSIF THIS^.P_bError THEN
			_inst_intStep := 0;
			bRouterBusy := FALSE;
		END_IF
		
	30: // Parse results
		_intRet := STRING_TO_INT(_inst_strRet);
		IF _intRet > 0 THEN
			_bResult := TRUE;
			THIS^.M_LogMessage(_strEND_MSG);
			// DO ANY PARSING HERE
//			_inst_fbParams.M_LoadFromParameterList(_inst_arrOutputs);
//			bConnected := _inst_fbParams.M_ParseBool(_inst_fbParams.M_GetParameter('connected'));
//			THIS^.bConnected := bConnected;
			
		// Set error if command failed
		ELSE
			THIS^.M_SetError(_udintERROR_ID, _strERROR_MSG);
		END_IF
		
		// Go back to start
		_inst_intStep := 0;
END_CASE
M_Tare := _bResult;
intTareStep := _inst_intStep;
END_METHOD

(* This method returns the status of whether the screen on the device has been locked.
Once the screen is locked, this method must return TRUE*)
METHOD M_UnlockDisplay : BOOL
VAR_INPUT
END_VAR
VAR CONSTANT
	_strCOMMAND_NAME : T_MaxString	:= 'UnlockDisplay'; // Name of the API method
	_timeCOMMAND_TIMEOUT : TIME		:= T#2S; // Max time to receive API response
	_strSTART_MSG : T_MaxString		:= 'Unlocking Alicat Display'; // Prints when method starts
	_strEND_MSG : T_MaxString		:= 'Unlocked Alicat Display'; // Prints when method finishes
	_udintERROR_ID : UDINT			:= E_Alicat_Error.FailedToUnlockDisplay; // Error ID to set if command fails
	_strERROR_MSG : T_MaxString		:= 'Failed to unlock display!'; // Error message to set if command fails
END_VAR
VAR_INST
	_inst_arrParams: T_ApiParameterList; // Parameters array
	_inst_arrOutputs: T_ApiParameterList; // Outputs array
	_inst_strRet: T_ApiParamValue; // Return string from the router
	_inst_intStep: INT; // Current method step
	_inst_fbParams: FB_ApiParamBuilder; // Parameter builder FB
END_VAR
VAR
	_bComplete: BOOL; // True if the routing finishes
	_intRet: INT; // Return string converted to an integer
	_bResult : BOOL; // Output of the method
END_VAR
_inst_intStep := intUnlockDisplayStep;
bUnlockDisplayBusy := TRUE;

_bResult := FALSE;
CASE _inst_intStep OF
	0: // Wait for no error and router not busy
		IF NOT THIS^.P_bError AND NOT bRouterBusy THEN
			bRouterBusy := TRUE;
			_inst_intStep := _inst_intStep + 10;
		END_IF
		
	10: // Initialize parameters
		THIS^.M_LogMessage(_strSTART_MSG);
		_inst_fbParams.M_ClearParameters();
		// ADD ANY PARAMETERS HERE
		_inst_fbParams.M_OutputToParameterList(_inst_arrParams);
		_inst_intStep := _inst_intStep + 10;
		
	20: // Route the command
		_bComplete := M_RouterHelper(
			_in_strMethodName := _strCOMMAND_NAME, 
			_in_timeTimeout := _timeCOMMAND_TIMEOUT,
			_inout_arrParams := _inst_arrParams,
			_inout_arrOutputs := _inst_arrOutputs,
			_out_strReturnValue=>_inst_strRet);
		
		// If route completed, move to next step
		IF _bComplete THEN
			_inst_intStep := _inst_intStep + 10;
			bRouterBusy := FALSE;
		ELSIF THIS^.P_bError THEN
			_inst_intStep := 0;
			bRouterBusy := FALSE;
		END_IF
		
	30: // Parse results
		_intRet := STRING_TO_INT(_inst_strRet);
		IF _intRet > 0 THEN
			_bResult := TRUE;
			THIS^.M_LogMessage(_strEND_MSG);
			// DO ANY PARSING HERE
//			_inst_fbParams.M_LoadFromParameterList(_inst_arrOutputs);
//			bConnected := _inst_fbParams.M_ParseBool(_inst_fbParams.M_GetParameter('connected'));
//			THIS^.bConnected := bConnected;
			
		// Set error if command failed
		ELSE
			THIS^.M_SetError(_udintERROR_ID, _strERROR_MSG);
		END_IF
		
		// Go back to start
		_inst_intStep := 0;
END_CASE
M_UnlockDisplay := _bResult;
intUnlockDisplayStep := _inst_intStep;
END_METHOD

(* This method should establish any external connections required to use the
	functions of the device, and return TRUE and set P_bConnected to TRUE once
	connected. *)
METHOD M_Connect : BOOL
VAR CONSTANT
	_strCOMMAND_NAME : T_MaxString	:= 'Connect'; // Name of the API method
	_timeCOMMAND_TIMEOUT : TIME		:= T#100S; // Max time to receive API response
	_strSTART_MSG : T_MaxString		:= 'Connecting'; // Prints when method starts
	_strEND_MSG : T_MaxString		:= 'Connected'; // Prints when method finishes
	_udintERROR_ID : UDINT			:= E_Alicat_Error.FailedToConnect; // Error ID to set if command fails
	_strERROR_MSG : T_MaxString		:= 'Failed to connect to Flow Meter!'; // Error message to set if command fails
END_VAR
VAR_INST
	_inst_arrParams: T_ApiParameterList; // Parameters array
	_inst_arrOutputs: T_ApiParameterList; // Outputs array
	_inst_strRet: T_ApiParamValue; // Return string from the router
	_inst_intStep: INT; // Current method step
	_inst_fbParams: FB_ApiParamBuilder; // Parameter builder FB
END_VAR
VAR
	_bComplete: BOOL; // True if the routing finishes
	_intRet: INT; // Return string converted to an integer
	_bResult : BOOL; // Output of the method
END_VAR
_inst_intStep := intConnectStep;
bConnectBusy  := TRUE;

_bResult := FALSE;
CASE _inst_intStep OF
	0: // Wait for no error and router not busy
		IF NOT THIS^.P_bError AND NOT bRouterBusy THEN
			bRouterBusy := TRUE;
			_inst_intStep := _inst_intStep + 10;
		END_IF
		
	10: // Initialize parameters
		THIS^.M_LogMessage(_strSTART_MSG);
		_inst_fbParams.M_ClearParameters();
		// ADD ANY PARAMETERS HERE
		_inst_fbParams.M_OutputToParameterList(_inst_arrParams);
		_inst_intStep := _inst_intStep + 10;
		
	20: // Route the command
		_bComplete := M_RouterHelper(
			_in_strMethodName := _strCOMMAND_NAME, 
			_in_timeTimeout := _timeCOMMAND_TIMEOUT,
			_inout_arrParams := _inst_arrParams,
			_inout_arrOutputs := _inst_arrOutputs,
			_out_strReturnValue=>_inst_strRet);
		
		// If route completed, move to next step
		IF _bComplete THEN
			_inst_intStep := _inst_intStep + 10;
			bRouterBusy := FALSE;
		ELSIF THIS^.P_bError THEN
			_inst_intStep := 0;
			bRouterBusy := FALSE;
		END_IF
		
	30: // Parse results
		_intRet := STRING_TO_INT(_inst_strRet);
		IF _intRet > 0 THEN
			_bResult := TRUE;
			THIS^.M_LogMessage(_strEND_MSG);
			// DO ANY PARSING HERE
			bConnected := TRUE;
			
		// Set error if command failed
		ELSE
			THIS^.M_SetError(_udintERROR_ID, _strERROR_MSG);
		END_IF
		
		// Go back to start
		_inst_intStep := 0;
END_CASE
M_Connect := _bResult;
intConnectStep := _inst_intStep;
END_METHOD

(* This method should break any connections established by M_Connect. It should
	immediately set P_bConnected to false unless all connections are known to
	be still active, and return TRUE once those connections are all fully
	disconnected. *)
METHOD M_Disconnect : BOOL
VAR CONSTANT
	_strCOMMAND_NAME : T_MaxString	:= 'Disconnect'; // Name of the API method
	_timeCOMMAND_TIMEOUT : TIME		:= T#30S; // Max time to receive API response
	_strSTART_MSG : T_MaxString		:= 'Disconnecting'; // Prints when method starts
	_strEND_MSG : T_MaxString		:= 'Disconnected'; // Prints when method finishes
	_udintERROR_ID : UDINT			:= E_Alicat_Error.FailedToDisconnect; // Error ID to set if command fails
	_strERROR_MSG : T_MaxString		:= 'Failed to disconnect from Flow Meter!'; // Error message to set if command fails
END_VAR
VAR_INST
	_inst_arrParams: T_ApiParameterList; // Parameters array
	_inst_arrOutputs: T_ApiParameterList; // Outputs array
	_inst_strRet: T_ApiParamValue; // Return string from the router
	_inst_intStep: INT; // Current method step
	_inst_fbParams: FB_ApiParamBuilder; // Parameter builder FB
END_VAR
VAR
	_bComplete: BOOL; // True if the routing finishes
	_intRet: INT; // Return string converted to an integer
	_bResult : BOOL; // Output of the method
END_VAR
_inst_intStep 	:= intDisconnectStep;
bDisconnectBusy := TRUE;

_bResult := FALSE;
CASE _inst_intStep OF
	0: // Wait for no error and router not busy
		IF NOT THIS^.P_bError AND NOT bRouterBusy THEN
			bRouterBusy := TRUE;
			_inst_intStep := _inst_intStep + 10;
		END_IF
		
	10: // Initialize parameters
		THIS^.M_LogMessage(_strSTART_MSG);
		_inst_fbParams.M_ClearParameters();
		// ADD ANY PARAMETERS HERE
		_inst_fbParams.M_OutputToParameterList(_inst_arrParams);
		_inst_intStep := _inst_intStep + 10;
		
	20: // Route the command
		_bComplete := M_RouterHelper(
			_in_strMethodName := _strCOMMAND_NAME, 
			_in_timeTimeout := _timeCOMMAND_TIMEOUT,
			_inout_arrParams := _inst_arrParams,
			_inout_arrOutputs := _inst_arrOutputs,
			_out_strReturnValue=>_inst_strRet);
		
		// If route completed, move to next step
		IF _bComplete THEN
			_inst_intStep := _inst_intStep + 10;
			bRouterBusy := FALSE;
		ELSIF THIS^.P_bError THEN
			_inst_intStep := 0;
			bRouterBusy := FALSE;
		END_IF
		
	30: // Parse results
		_intRet := STRING_TO_INT(_inst_strRet);
		IF _intRet > 0 THEN
			_bResult := TRUE;
			THIS^.M_LogMessage(_strEND_MSG);
			// DO ANY PARSING HERE
			bConnected := FALSE;
			
		// Set error if command failed
		ELSE
			THIS^.M_SetError(_udintERROR_ID, _strERROR_MSG);
		END_IF
		
		// Go back to start
		_inst_intStep := 0;
END_CASE
M_Disconnect := _bResult;
intDisconnectStep := _inst_intStep;
END_METHOD

(* This method should explicitly check the connection status of the device.
	Once the connection status is known, this method should return TRUE.
	If this method fails, P_bConnected should be set to FALSE since the device
	is not absolutely known to still be connected. *)
METHOD M_GetConnectStatus : BOOL
VAR_OUTPUT
	(* This should return TRUE if all connections required to make the device
		function properly are known to be connected, and FALSE otherwise. *)
	bConnected	: BOOL;
END_VAR
bConnected := P_bConnected;
M_GetConnectStatus := TRUE;
THIS^.M_LogWarning('Get connect status not implemented in FB_FlowMeter!');
END_METHOD

(* This property should be TRUE while any method in this interface is actively
	executing, or FALSE otherwise. *)
PROPERTY P_bConnectBusy : BOOL
GET
END_GET
END_PROPERTY

(* This should be set to TRUE if M_Connect is successful or M_GetConnectStatus
	determines the device to be connected, and set to FALSE if M_Disconnect is
	called at all, M_GetConnectStatus fails, or M_GetConnectStatus determines
	the device to be not connected. *)
PROPERTY P_bConnected : BOOL
GET
END_GET
END_PROPERTY

PROPERTY P_strDescription : Sensata_Common.T_MaxString
GET
END_GET
END_PROPERTY

PROPERTY P_strMake : Sensata_Common.T_MaxString
GET
END_GET
END_PROPERTY

PROPERTY P_strModel : Sensata_Common.T_MaxString
GET
END_GET
END_PROPERTY

PROPERTY P_strVersion : Sensata_Common.T_MaxString
GET
END_GET
END_PROPERTY

(* This method returns the Pressure Value from the Alicat Flow Meter.
Once the Pressure value is obtained, this method must return TRUE*)
METHOD M_GetPressure : BOOL
VAR_OUTPUT
	(*_output/input_datatypeName*)
	_out_lrealPressure	    : LREAL;
//	_out_lrealTotalizedFlow : LREAL;
//	_out_lrealMassFlowRate	: LREAL;
//	_out_lrealVolFlowRate   : LREAL;
END_VAR
VAR CONSTANT
	_strCOMMAND_NAME : T_MaxString	:= 'GetPressure'; // Name of the API method
	_timeCOMMAND_TIMEOUT : TIME		:= T#5S; // Max time to receive API response
	_strSTART_MSG : T_MaxString		:= 'Reading Pressure Value'; // Prints when method starts
	_strEND_MSG : T_MaxString		:= 'Pressure Read'; // Prints when method finishes
	_udintERROR_ID : UDINT			:= E_Alicat_Error.FailedToReadSerialData; // Error ID to set if command fails
	_strERROR_MSG : T_MaxString		:= 'Failed to read serial data and hence pressure!'; // Error message to set if command fails
END_VAR
VAR_INST
	_inst_arrParams: T_ApiParameterList; // Parameters array
	_inst_arrOutputs: T_ApiParameterList; // Outputs array
	_inst_strRet: T_ApiParamValue; // Return string from the router
	_inst_intStep: INT; // Current method step
	_inst_fbParams: FB_ApiParamBuilder; // Parameter builder FB
END_VAR
VAR
	_bComplete: BOOL; // True if the routing finishes
	_intRet: INT; // Return string converted to an integer
	_bResult : BOOL; // Output of the method
END_VAR
_inst_intStep 	 := intGetPressureStep;
bGetPressureBusy := TRUE;

_bResult := FALSE;
CASE _inst_intStep OF
	0: // Wait for no error and router not busy
		IF NOT THIS^.P_bError AND NOT bRouterBusy THEN
			bRouterBusy := TRUE;
			_inst_intStep := _inst_intStep + 10;
		END_IF
		
	10: // Initialize parameters
		THIS^.M_LogMessage(_strSTART_MSG);
		_inst_fbParams.M_ClearParameters();
		// ADD ANY PARAMETERS HERE
		_inst_fbParams.M_OutputToParameterList(_inst_arrParams);
		_inst_intStep := _inst_intStep + 10;
		
	20: // Route the command
		_bComplete := M_RouterHelper(
			_in_strMethodName := _strCOMMAND_NAME, 
			_in_timeTimeout := _timeCOMMAND_TIMEOUT,
			_inout_arrParams := _inst_arrParams,
			_inout_arrOutputs := _inst_arrOutputs,
			_out_strReturnValue=>_inst_strRet);
		
		// If route completed, move to next step
		IF _bComplete THEN
			_inst_intStep := _inst_intStep + 10;
			bRouterBusy := FALSE;
		ELSIF THIS^.P_bError THEN
			_inst_intStep := 0;
			bRouterBusy := FALSE;
		END_IF
		
	30: // Parse results
		_intRet := STRING_TO_INT(_inst_strRet);
		IF _intRet > 0 THEN
			_bResult := TRUE;
			THIS^.M_LogMessage(_strEND_MSG);
			// DO ANY PARSING HERE
			_out_lrealPressure := _inst_fbParams.M_ParseDouble(_inst_fbParams.M_GetParameter('Pressure'));
//			_inst_fbParams.M_LoadFromParameterList(_inst_arrOutputs);
//			bEnabled := _inst_fbParams.M_ParseBool(_inst_fbParams.M_GetParameter('enabled'));
//			THIS^.bEnabled := bEnabled;			
			
		// Set error if command failed
		ELSE
			THIS^.M_SetError(_udintERROR_ID, _strERROR_MSG);
		END_IF
		
		// Go back to start
		_inst_intStep := 0;
END_CASE
M_GetPressure := _bResult;
intGetPressureStep := _inst_intStep;
END_METHOD

ACTION A_CommandRecovery:
IF NOT bGetPressureBusy AND intGetPressureStep > 0 THEN
	intGetPressureStep := 0;
	bRouterBusy := FALSE;
	THIS^.M_LogWarning('Get Pressure ended prematurely!');
END_IF
bGetPressureBusy := FALSE;

IF NOT bConnectBusy AND intConnectStep > 0 THEN
	intConnectStep := 0;
	bRouterBusy := FALSE;
	THIS^.M_LogWarning('Connect ended prematurely!');
END_IF
bConnectBusy := FALSE;

IF NOT bDisconnectBusy AND intDisconnectStep > 0 THEN
	intDisconnectStep := 0;
	bRouterBusy := FALSE;
	THIS^.M_LogWarning('Disconnect ended prematurely!');
END_IF
bDisconnectBusy := FALSE;

